  MoveL 6472 to (3.7, 324.47, -39.12) mm, rotated rx -180 ry 0 rz 0.01 deg; joints [44.471, -46.671, 108.236, -132.07, 70.721, 160.68]
  MoveL 6473 to (-1.54, 328.5, -39.37) mm, rotated rx 180 ry 0 rz 0.01 deg; joints [44.44, -46.388, 107.644, -132.02, 70.503, 160.447]
  MoveL 6474 to (0.05, 334.91, -39.61) mm, rotated rx -180 ry 0 rz 0.01 deg; joints [44.663, -46.238, 107.338, -131.758, 70.479, 160.247]
  MoveL 6475 to (6.56, 336.02, -39.86) mm, rotated rx 180 ry 0 rz 0.01 deg; joints [44.874, -46.386, 107.685, -131.602, 70.686, 160.333]
  MoveL 6476 to (10.19, 330.5, -40.1) mm, rotated rx -180 ry 0 rz 0.01 deg; joints [44.821, -46.638, 108.266, -131.74, 70.887, 160.611]
  MoveL 6477 to (6.58, 324.97, -40.35) mm, rotated rx -180 ry 0 rz 0.01 deg; joints [44.566, -46.676, 108.384, -132.014, 70.85, 160.76]
  MoveL 6478 to (0.07, 326.05, -40.59) mm, rotated rx 180 ry 0 rz 0.01 deg; joints [44.416, -46.439, 107.896, -132.097, 70.629, 160.613]
  MoveL 6479 to (-1.55, 332.45, -40.83) mm, rotated rx -180 ry 0 rz 0.01 deg; joints [44.551, -46.195, 107.385, -131.893, 70.498, 160.357]
  MoveL 6480 to (3.67, 336.5, -41.08) mm, rotated rx 180 ry 0 rz 0.01 deg; joints [44.808, -46.221, 107.462, -131.652, 70.625, 160.31]
  MoveL 6481 to (9.47, 333.34, -41.32) mm, rotated rx 180 ry 0 rz 0.01 deg; joints [44.881, -46.469, 108.034, -131.664, 70.865, 160.541]
  MoveL 6482 to (8.9, 326.76, -41.57) mm, rotated rx -180 ry 0 rz 0.01 deg; joints [44.681, -46.627, 108.413, -131.919, 70.943, 160.783]
  MoveL 6483 to (2.64, 324.65, -41.81) mm, rotated rx -180 ry 0 rz 0.01 deg; joints [44.448, -46.489, 108.144, -132.116, 70.773, 160.758]
  MoveL 6484 to (-1.8, 329.53, -42.05) mm, rotated rx -180 ry 0 rz 0.01 deg; joints [44.463, -46.205, 107.548, -132.02, 70.569, 160.507]
  MoveL 6485 to (0.89, 335.56, -42.3) mm, rotated rx -180 ry 0 rz 0.01 deg; joints [44.706, -46.1, 107.337, -131.752, 70.586, 160.342]
  MoveL 6486 to (7.49, 335.51, -42.54) mm, rotated rx -180 ry 0 rz 0.01 deg; joints [44.887, -46.283, 107.763, -131.636, 70.812, 160.472]
  MoveL 6487 to (10.09, 329.44, -42.79) mm, rotated rx 180 ry 0 rz 0.01 deg; joints [44.79, -46.519, 108.314, -131.814, 70.986, 160.753]
  MoveL 6488 to (5.57, 324.62, -43.03) mm, rotated rx -180 ry 0 rz 0.01 deg; joints [44.529, -46.51, 108.327, -132.078, 70.91, 160.858]
  MoveL 6489 to (-0.65, 326.84, -43.27) mm, rotated rx 180 ry 0 rz 0.01 deg; joints [44.419, -46.25, 107.786, -132.114, 70.683, 160.674]
  MoveL 6490 to (-1.12, 333.42, -43.52) mm, rotated rx 180 ry 0 rz 0.01 deg; joints [44.591, -46.035, 107.338, -131.883, 70.588, 160.432]
  MoveL 6491 to (4.73, 336.49, -43.76) mm, rotated rx -180 ry 0 rz 0.01 deg; joints [44.838, -46.108, 107.517, -131.666, 70.748, 160.433]
  MoveL 6492 to (9.89, 332.36, -44.01) mm, rotated rx -180 ry 0 rz 0.01 deg; joints [44.866, -46.364, 108.109, -131.725, 70.98, 160.688]
  MoveL 6493 to (8.17, 325.99, -44.25) mm, rotated rx 180 ry 0 rz 0.01 deg; joints [44.64, -46.481, 108.401, -131.995, 71.018, 160.902]
  MoveL 6494 to (1.64, 325, -44.49) mm, rotated rx -180 ry 0 rz 0.01 deg; joints [44.431, -46.303, 108.043, -132.155, 70.824, 160.83]
  MoveL 6495 to (-1.88, 330.59, -44.74) mm, rotated rx -180 ry 0 rz 0.01 deg; joints [44.492, -46.027, 107.461, -132.016, 70.64, 160.569]
  MoveL 6496 to (1.83, 336.06, -44.98) mm, rotated rx 180 ry 0 rz 0.01 deg; joints [44.747, -45.968, 107.352, -131.75, 70.698, 160.444]
  MoveL 6497 to (8.33, 334.84, -45.23) mm, rotated rx 180 ry 0 rz 0.01 deg; joints [44.893, -46.181, 107.845, -131.678, 70.936, 160.616]
  MoveL 6498 to (9.82, 328.41, -45.47) mm, rotated rx 180 ry 0 rz 0.01 deg; joints [44.754, -46.394, 108.347, -131.89, 71.08, 160.89]
  MoveL 6499 to (4.52, 324.47, -45.71) mm, rotated rx -180 ry 0 rz 0.01 deg; joints [44.496, -46.337, 108.255, -132.136, 70.967, 160.949]
  MoveL 6500 to (-1.22, 327.74, -45.96) mm, rotated rx -180 ry 0 rz 0.01 deg; joints [44.43, -46.062, 107.678, -132.124, 70.741, 160.734]
  MoveL 6501 to (-0.52, 334.31, -46.2) mm, rotated rx 180 ry 0 rz 0.01 deg; joints [44.633, -45.883, 107.306, -131.872, 70.683, 160.513]
  MoveL 6502 to (5.78, 336.3, -46.45) mm, rotated rx -180 ry 0 rz 0.01 deg; joints [44.863, -45.998, 107.582, -131.687, 70.872, 160.563]
  MoveL 6503 to (10.13, 331.32, -46.69) mm, rotated rx 180 ry 0 rz 0.01 deg; joints [44.845, -46.254, 108.175, -131.792, 71.09, 160.835]
  MoveL 6504 to (7.31, 325.35, -46.93) mm, rotated rx 180 ry 0 rz 0.01 deg; joints [44.599, -46.327, 108.372, -132.067, 71.087, 161.013]
  MoveL 6505 to (0.71, 325.53, -47.18) mm, rotated rx 180 ry 0 rz 0.01 deg; joints [44.422, -46.115, 107.935, -132.185, 70.875, 160.897]
  MoveL 6506 to (-1.76, 331.65, -47.42) mm, rotated rx 180 ry 0 rz 0.01 deg; joints [44.525, -45.855, 107.387, -132.008, 70.717, 160.635]
  MoveL 6507 to (2.85, 336.38, -47.67) mm, rotated rx -180 ry 0 rz 0.01 deg; joints [44.785, -45.844, 107.382, -131.753, 70.814, 160.553]
  MoveL 6508 to (9.03, 334.04, -47.91) mm, rotated rx -180 ry 0 rz 0.01 deg; joints [44.891, -46.078, 107.926, -131.728, 71.057, 160.761]
  MoveL 6509 to (9.36, 327.44, -48.15) mm, rotated rx -180 ry 0 rz 0.01 deg; joints [44.715, -46.261, 108.364, -131.966, 71.166, 161.02]
  MoveL 6510 to (3.45, 324.5, -48.4) mm, rotated rx 180 ry 0 rz 0.01 deg; joints [44.469, -46.158, 108.17, -132.188, 71.02, 161.031]
  MoveL 6511 to (-1.62, 328.73, -48.64) mm, rotated rx -180 ry 0 rz 0.01 deg; joints [44.448, -45.876, 107.575, -132.128, 70.802, 160.792]
  MoveL 6512 to (0.23, 335.07, -48.89) mm, rotated rx 180 ry 0 rz 0.01 deg; joints [44.676, -45.738, 107.29, -131.864, 70.785, 160.6]
  MoveL 6513 to (6.78, 335.92, -49.13) mm, rotated rx 180 ry 0 rz 0.01 deg; joints [44.881, -45.893, 107.655, -131.715, 70.997, 160.698]
  MoveL 6514 to (10.18, 330.26, -49.38) mm, rotated rx 180 ry 0 rz 0.01 deg; joints [44.818, -46.139, 108.231, -131.862, 71.195, 160.978]
  MoveL 6515 to (6.36, 324.87, -49.62) mm, rotated rx -180 ry 0 rz 0.01 deg; joints [44.56, -46.165, 108.325, -132.134, 71.151, 161.117]
  MoveL 6516 to (-0.11, 326.22, -49.86) mm, rotated rx 180 ry 0 rz 0.01 deg; joints [44.419, -45.925, 107.824, -132.208, 70.926, 160.959]
  MoveL 6517 to (-1.47, 332.68, -50.11) mm, rotated rx -180 ry 0 rz 0.01 deg; joints [44.563, -45.689, 107.325, -131.997, 70.801, 160.704]
  MoveL 6518 to (3.91, 336.51, -50.35) mm, rotated rx -180 ry 0 rz 0.01 deg; joints [44.819, -45.725, 107.426, -131.761, 70.934, 160.67]
  MoveL 6519 to (9.58, 333.13, -50.6) mm, rotated rx 180 ry 0 rz 0.01 deg; joints [44.882, -45.974, 108.003, -131.783, 71.175, 160.908]
  MoveL 6520 to (8.75, 326.57, -50.84) mm, rotated rx 180 ry 0 rz 0.01 deg; joints [44.675, -46.12, 108.363, -132.042, 71.246, 161.144]
  MoveL 6521 to (2.41, 324.71, -51.08) mm, rotated rx 180 ry 0 rz 0.01 deg; joints [44.447, -45.974, 108.073, -132.231, 71.071, 161.106]
  MoveL 6522 to (-1.84, 329.77, -51.33) mm, rotated rx 180 ry 0 rz 0.01 deg; joints [44.472, -45.694, 107.479, -132.126, 70.868, 160.852]
  MoveL 6523 to (1.1, 335.69, -51.57) mm, rotated rx 180 ry 0 rz 0.01 deg; joints [44.718, -45.6, 107.291, -131.858, 70.892, 160.695]
  MoveL 6524 to (7.69, 335.37, -51.82) mm, rotated rx 180 ry 0 rz 0.01 deg; joints [44.892, -45.789, 107.733, -131.751, 71.122, 160.837]
  MoveL 6525 to (10.05, 329.2, -52.06) mm, rotated rx 180 ry 0 rz 0.01 deg; joints [44.785, -46.018, 108.273, -131.936, 71.293, 161.118]
  MoveL 6526 to (5.34, 324.57, -52.3) mm, rotated rx 180 ry 0 rz 0.01 deg; joints [44.524, -45.997, 108.263, -132.197, 71.209, 161.211]
  MoveL 6527 to (-0.79, 327.03, -52.55) mm, rotated rx -180 ry 0 rz 0.01 deg; joints [44.425, -45.735, 107.712, -132.222, 70.98, 161.018]
  MoveL 6528 to (-0.99, 333.63, -52.79) mm, rotated rx -180 ry 0 rz 0.01 deg; joints [44.604, -45.53, 107.279, -131.986, 70.891, 160.779]
  MoveL 6529 to (4.97, 336.46, -53.04) mm, rotated rx -180 ry 0 rz 0.01 deg; joints [44.848, -45.612, 107.482, -131.776, 71.057, 160.793]
  MoveL 6530 to (9.96, 332.13, -53.28) mm, rotated rx 180 ry 0 rz 0.01 deg; joints [44.865, -45.866, 108.075, -131.845, 71.289, 161.054]
  MoveL 6531 to (7.98, 325.83, -53.52) mm, rotated rx 180 ry 0 rz 0.01 deg; joints [44.634, -45.972, 108.346, -132.116, 71.32, 161.26]
  MoveL 6532 to (1.42, 325.11, -53.77) mm, rotated rx 180 ry 0 rz 0.01 deg; joints [44.432, -45.787, 107.968, -132.267, 71.12, 161.176]
  MoveL 6533 to (-1.87, 330.84, -54.01) mm, rotated rx 180 ry 0 rz 0.01 deg; joints [44.502, -45.517, 107.393, -132.12, 70.94, 160.913]
  MoveL 6534 to (2.06, 336.15, -54.26) mm, rotated rx -180 ry 0 rz 0.01 deg; joints [44.759, -45.469, 107.307, -131.856, 71.005, 160.798]
  MoveL 6535 to (8.5, 334.67, -54.5) mm, rotated rx 180 ry 0 rz 0.01 deg; joints [44.896, -45.685, 107.812, -131.794, 71.246, 160.98]
  MoveL 6536 to (8.17, 335.16, -54.5) mm, rotated rx -180 ry 0 rz 0.01 deg; joints [44.9, -45.662, 107.76, -131.782, 71.228, 160.956]
  MoveL 6537 to (9.9, 336.02, -54.5) mm, rotated rx 180 ry 0 rz 0.01 deg; joints [44.973, -45.688, 107.816, -131.718, 71.273, 160.956]
  MoveL 6538 to (10.07, 335.56, -54.5) mm, rotated rx -180 ry 0 rz 0.01 deg; joints [44.965, -45.706, 107.857, -131.732, 71.285, 160.976]
  MoveL 6539 to (10.27, 334.35, -54.5) mm, rotated rx -180 ry 0 rz 0.01 deg; joints [44.936, -45.745, 107.946, -131.772, 71.308, 161.025]
  MoveL 6540 to (10.27, 32.01, -54.5) mm, rotated rx 180 ry 0 rz 0.01 deg; joints [35.147, -52.794, 124.522, -143.55, 75.758, 170.644]
  MoveL 6541 to (9.41, 35.75, -54.5) mm, rotated rx -180 ry 0 rz 0.01 deg; joints [35.264, -52.7, 124.291, -143.411, 75.67, 170.53]
  MoveL 6542 to (9.3, 36.12, -54.5) mm, rotated rx 180 ry 0 rz 0.01 deg; joints [35.275, -52.689, 124.267, -143.398, 75.66, 170.518]
  MoveL 6543 to (8.81, 37.5, -54.5) mm, rotated rx -180 ry 0 rz 0.01 deg; joints [35.313, -52.65, 124.17, -143.351, 75.621, 170.473]
  MoveL 6544 to (8.66, 37.84, -54.5) mm, rotated rx 180 ry 0 rz 0.01 deg; joints [35.321, -52.639, 124.145, -143.34, 75.611, 170.462]
  MoveL 6545 to (8, 39.21, -54.5) mm, rotated rx -180 ry 0 rz 0.01 deg; joints [35.355, -52.595, 124.036, -143.296, 75.566, 170.414]
  MoveL 6546 to (7.87, 39.46, -54.5) mm, rotated rx -180 ry 0 rz 0.01 deg; joints [35.36, -52.586, 124.017, -143.289, 75.558, 170.405]
  MoveL 6547 to (2.64, 48.31, -54.5) mm, rotated rx -180 ry 0 rz 0.01 deg; joints [35.549, -52.271, 123.255, -143.028, 75.238, 170.078]
  MoveL 6548 to (2.37, 48.71, -54.5) mm, rotated rx 180 ry 0 rz 0.01 deg; joints [35.556, -52.255, 123.218, -143.017, 75.222, 170.063]
  MoveL 6549 to (1.13, 50.25, -54.5) mm, rotated rx -180 ry 0 rz 0.01 deg; joints [35.58, -52.191, 123.063, -142.978, 75.154, 170]
  MoveL 6550 to (0.8, 50.61, -54.5) mm, rotated rx 180 ry 0 rz 0.01 deg; joints [35.585, -52.175, 123.025, -142.97, 75.137, 169.985]
  MoveL 6551 to (0, 51.35, -54.5) mm, rotated rx 180 ry 0 rz 0.01 deg; joints [35.591, -52.138, 122.937, -142.955, 75.098, 169.952]
  MoveL 6552 to (-1.84, 53.24, -54.5) mm, rotated rx 180 ry 0 rz 0.01 deg; joints [35.612, -52.049, 122.725, -142.915, 75.004, 169.869]
  MoveL 6553 to (-1.94, 53.34, -54.5) mm, rotated rx -180 ry 0 rz 0.01 deg; joints [35.613, -52.044, 122.713, -142.912, 74.999, 169.865]
  MoveL 6554 to (-4.34, 55.6, -54.5) mm, rotated rx 180 ry 0 rz 0.01 deg; joints [35.632, -51.932, 122.447, -142.868, 74.88, 169.763]
  MoveL 6555 to (-4.53, 55.76, -54.5) mm, rotated rx -180 ry 0 rz 0.01 deg; joints [35.633, -51.924, 122.427, -142.865, 74.87, 169.755]
  MoveL 6556 to (-7.2, 57.93, -54.5) mm, rotated rx -180 ry 0 rz 0.01 deg; joints [35.643, -51.805, 122.146, -142.829, 74.743, 169.651]
  MoveL 6557 to (-7.35, 58.05, -54.5) mm, rotated rx 180 ry 0 rz 0.01 deg; joints [35.643, -51.799, 122.13, -142.827, 74.735, 169.645]
  MoveL 6558 to (-117.5, 137.2, -54.5) mm, rotated rx 180 ry 0 rz 0.01 deg; joints [35.648, -46.798, 110.617, -141.535, 69.59, 165.45]
  MoveL 6559 to (-117.96, 137.48, -54.5) mm, rotated rx -180 ry 0 rz 0.01 deg; joints [35.647, -46.777, 110.57, -141.531, 69.569, 165.433]
  MoveL 6560 to (-119.42, 138.21, -54.5) mm, rotated rx 180 ry 0 rz 0.01 deg; joints [35.636, -46.714, 110.427, -141.523, 69.504, 165.385]
  MoveL 6561 to (-120.06, 138.45, -54.5) mm, rotated rx -180 ry 0 rz 0.01 deg; joints [35.629, -46.688, 110.369, -141.523, 69.477, 165.366]
  MoveL 6562 to (-121.51, 138.84, -54.5) mm, rotated rx -180 ry 0 rz 0.01 deg; joints [35.608, -46.632, 110.245, -141.528, 69.417, 165.328]
  MoveL 6563 to (-122.11, 138.94, -54.5) mm, rotated rx -180 ry 0 rz 0.01 deg; joints [35.597, -46.61, 110.196, -141.533, 69.393, 165.314]
  MoveL 6564 to (-123.56, 139.06, -54.5) mm, rotated rx -180 ry 0 rz 0.01 deg; joints [35.567, -46.56, 110.085, -141.549, 69.337, 165.285]
  MoveL 6565 to (-124.2, 139.05, -54.5) mm, rotated rx -180 ry 0 rz 0.01 deg; joints [35.552, -46.54, 110.039, -141.559, 69.313, 165.274]
  MoveL 6566 to (-126.74, 138.78, -54.5) mm, rotated rx 180 ry 0 rz 0.01 deg; joints [35.484, -46.463, 109.87, -141.607, 69.222, 165.238]
  MoveL 6567 to (-127.23, 138.69, -54.5) mm, rotated rx -180 ry 0 rz 0.01 deg; joints [35.47, -46.449, 109.839, -141.618, 69.205, 165.232]
  MoveL 6568 to (-129.41, 138.12, -54.5) mm, rotated rx -180 ry 0 rz 0.01 deg; joints [35.401, -46.391, 109.711, -141.672, 69.131, 165.211]
  MoveL 6569 to (-129.67, 138.04, -54.5) mm, rotated rx 180 ry 0 rz 0.01 deg; joints [35.392, -46.384, 109.696, -141.679, 69.122, 165.209]
  MoveL 6570 to (-131.12, 137.53, -54.5) mm, rotated rx 180 ry 0 rz 0.01 deg; joints [35.342, -46.348, 109.617, -141.72, 69.074, 165.199]
  MoveL 6571 to (-131.37, 137.43, -54.5) mm, rotated rx 180 ry 0 rz 0.01 deg; joints [35.333, -46.342, 109.603, -141.728, 69.066, 165.198]
  MoveL 6572 to (-134.37, 136.1, -54.5) mm, rotated rx 180 ry 0 rz 0.01 deg; joints [35.221, -46.273, 109.453, -141.825, 68.971, 165.187]
  MoveL 6573 to (-134.69, 135.94, -54.5) mm, rotated rx -180 ry 0 rz 0.01 deg; joints [35.208, -46.266, 109.439, -141.836, 68.961, 165.187]
  MoveL 6574 to (-171.12, 114.98, -54.5) mm, rotated rx 180 ry 0 rz 0.01 deg; joints [33.707, -45.509, 107.806, -143.175, 67.848, 165.2]
  MoveL 6575 to (-171.78, 114.49, -54.5) mm, rotated rx 180 ry 0 rz 0.01 deg; joints [33.676, -45.497, 107.781, -143.204, 67.829, 165.204]
  MoveL 6576 to (-172.53, 113.77, -54.5) mm, rotated rx -180 ry 0 rz 0.01 deg; joints [33.636, -45.487, 107.761, -143.243, 67.809, 165.213]
  MoveC 6577 to (-172.87, 113.39, -54.5) mm, rotated rx -180 ry 0 rz 0.01 deg; joints [33.617, -45.484, 107.754, -143.262, 67.801, 165.219] to (-173.15, 112.97, -54.5) mm, rotated rx 180 ry 0 rz 0.01 deg; joints [33.597, -45.483, 107.754, -143.283, 67.796, 165.227]
  MoveL 6578 to (-173.64, 112.08, -54.5) mm, rotated rx 180 ry 0 rz 0.01 deg; joints [33.557, -45.486, 107.761, -143.325, 67.789, 165.246]
  MoveC 6579 to (-173.86, 111.61, -54.5) mm, rotated rx 180 ry 0 rz 0.01 deg; joints [33.537, -45.489, 107.768, -143.347, 67.787, 165.257] to (-174, 111.11, -54.5) mm, rotated rx -180 ry 0 rz 0.01 deg; joints [33.517, -45.495, 107.782, -143.37, 67.788, 165.27]
  MoveL 6580 to (-174.22, 110.02, -54.5) mm, rotated rx 180 ry 0 rz 0.01 deg; joints [33.477, -45.511, 107.82, -143.417, 67.794, 165.301]
  MoveC 6581 to (-174.29, 109.49, -54.5) mm, rotated rx 180 ry 0 rz 0.01 deg; joints [33.458, -45.52, 107.841, -143.44, 67.798, 165.316] to (-174.27, 108.95, -54.5) mm, rotated rx -180 ry 0 rz 0.01 deg; joints [33.44, -45.532, 107.87, -143.461, 67.806, 165.333]
  MoveL 6582 to (-174.14, 107.86, -54.5) mm, rotated rx -180 ry 0 rz 0.01 deg; joints [33.408, -45.56, 107.933, -143.504, 67.826, 165.37]
  MoveC 6583 to (-174.03, 107.32, -54.5) mm, rotated rx -180 ry 0 rz 0.01 deg; joints [33.392, -45.576, 107.969, -143.525, 67.837, 165.389] to (-173.83, 106.8, -54.5) mm, rotated rx -180 ry 0 rz 0.01 deg; joints [33.379, -45.594, 108.009, -143.544, 67.852, 165.408]
  MoveL 6584 to (-173.32, 105.74, -54.5) mm, rotated rx -180 ry 0 rz 0.01 deg; joints [33.355, -45.634, 108.1, -143.581, 67.886, 165.45]
  MoveC 6585 to (-173.06, 105.29, -54.5) mm, rotated rx -180 ry 0 rz 0.01 deg; joints [33.346, -45.652, 108.142, -143.596, 67.903, 165.469] to (-172.73, 104.88, -54.5) mm, rotated rx 180 ry 0 rz 0.01 deg; joints [33.34, -45.673, 108.187, -143.609, 67.921, 165.488]
  MoveL 6586 to (-172.05, 104.16, -54.5) mm, rotated rx 180 ry 0 rz 0.01 deg; joints [33.331, -45.711, 108.273, -143.629, 67.957, 165.522]
  MoveL 6587 to (-171.28, 103.56, -54.5) mm, rotated rx -180 ry 0 rz 0.01 deg; joints [33.328, -45.75, 108.36, -143.644, 67.995, 165.554]
  MoveL 6588 to (-55.84, 36.98, -54.5) mm, rotated rx 180 ry 0 rz 0.01 deg; joints [33.667, -50.782, 119.826, -144.62, 73.292, 169.428]
  MoveL 6589 to (-63.76, 23.29, -54.5) mm, rotated rx 180 ry 0 rz 0.01 deg; joints [32.98, -50.8, 119.9, -145.332, 73.197, 169.672]
  MoveL 6590 to (-178.74, 89.79, -54.5) mm, rotated rx -180 ry 0 rz 0.01 deg; joints [32.71, -45.788, 108.472, -144.303, 67.887, 165.848]
  MoveL 6591 to (-179.27, 90.04, -54.5) mm, rotated rx 180 ry 0 rz 0.01 deg; joints [32.707, -45.765, 108.42, -144.299, 67.863, 165.831]
  MoveL 6592 to (-180.24, 90.4, -54.5) mm, rotated rx -180 ry 0 rz 0.01 deg; joints [32.698, -45.724, 108.329, -144.297, 67.82, 165.803]
  MoveC 6593 to (-180.73, 90.53, -54.5) mm, rotated rx 180 ry 0 rz 0.01 deg; joints [32.693, -45.704, 108.285, -144.297, 67.799, 165.79] to (-181.24, 90.6, -54.5) mm, rotated rx 180 ry 0 rz 0.01 deg; joints [32.684, -45.685, 108.244, -144.301, 67.778, 165.779]
  MoveL 6594 to (-182.28, 90.65, -54.5) mm, rotated rx -180 ry 0 rz 0.01 deg; joints [32.664, -45.649, 108.162, -144.311, 67.737, 165.759]
  MoveC 6595 to (-182.79, 90.64, -54.5) mm, rotated rx 180 ry 0 rz 0.01 deg; joints [32.652, -45.631, 108.124, -144.318, 67.716, 165.751] to (-183.29, 90.55, -54.5) mm, rotated rx -180 ry 0 rz 0.01 deg; joints [32.638, -45.616, 108.09, -144.328, 67.698, 165.745]
  MoveL 6596 to (-184.32, 90.28, -54.5) mm, rotated rx -180 ry 0 rz 0.01 deg; joints [32.608, -45.586, 108.025, -144.351, 67.661, 165.735]
  MoveC 6597 to (-184.81, 90.11, -54.5) mm, rotated rx 180 ry 0 rz 0.01 deg; joints [32.592, -45.573, 107.996, -144.364, 67.644, 165.732] to (-185.27, 89.87, -54.5) mm, rotated rx -180 ry 0 rz 0.01 deg; joints [32.574, -45.562, 107.973, -144.38, 67.629, 165.731]
  MoveL 6598 to (-186.19, 89.29, -54.5) mm, rotated rx 180 ry 0 rz 0.01 deg; joints [32.535, -45.543, 107.931, -144.415, 67.6, 165.733]
  MoveL 6599 to (-186.72, 88.88, -54.5) mm, rotated rx 180 ry 0 rz 0.01 deg; joints [32.51, -45.533, 107.911, -144.438, 67.585, 165.736]
  MoveL 6600 to (-186.93, 88.67, -54.5) mm, rotated rx 180 ry 0 rz 0.01 deg; joints [32.499, -45.53, 107.904, -144.449, 67.579, 165.739]
  MoveL 6601 to (-187.39, 88.14, -54.5) mm, rotated rx 180 ry 0 rz 0.01 deg; joints [32.471, -45.526, 107.896, -144.477, 67.568, 165.747]
  MoveL 6602 to (-188.03, 87.2, -54.5) mm, rotated rx 180 ry 0 rz 0.01 deg; joints [32.427, -45.523, 107.892, -144.523, 67.555, 165.765]
  MoveC 6603 to (-188.3, 86.74, -54.5) mm, rotated rx 180 ry 0 rz 0.01 deg; joints [32.406, -45.524, 107.894, -144.545, 67.551, 165.774] to (-188.48, 86.25, -54.5) mm, rotated rx -180 ry 0 rz 0.01 deg; joints [32.386, -45.527, 107.903, -144.568, 67.55, 165.786]
  MoveL 6604 to (-188.77, 85.29, -54.5) mm, rotated rx -180 ry 0 rz 0.01 deg; joints [32.347, -45.538, 107.928, -144.611, 67.551, 165.811]
  MoveL 6605 to (-188.91, 84.32, -54.5) mm, rotated rx 180 ry 0 rz 0.01 deg; joints [32.312, -45.553, 107.964, -144.653, 67.558, 165.838]
  MoveL 6606 to (-188.88, 42.24, -54.5) mm, rotated rx 180 ry 0 rz 0.01 deg; joints [30.889, -46.405, 109.934, -146.395, 68.114, 167.097]
  MoveL 6607 to (-188.87, 41.91, -54.5) mm, rotated rx -180 ry 0 rz 0.01 deg; joints [30.878, -46.412, 109.95, -146.409, 68.119, 167.107]
  MoveL 6608 to (-188.58, 39.01, -54.5) mm, rotated rx 180 ry 0 rz 0.01 deg; joints [30.784, -46.478, 110.104, -146.526, 68.169, 167.196]
  MoveL 6609 to (-188.54, 38.69, -54.5) mm, rotated rx 180 ry 0 rz 0.01 deg; joints [30.774, -46.486, 110.122, -146.539, 68.175, 167.206]
  MoveL 6610 to (-187.97, 35.79, -54.5) mm, rotated rx 180 ry 0 rz 0.01 deg; joints [30.686, -46.562, 110.296, -146.653, 68.235, 167.3]
  MoveL 6611 to (-187.88, 35.43, -54.5) mm, rotated rx 180 ry 0 rz 0.01 deg; joints [30.675, -46.572, 110.319, -146.666, 68.244, 167.312]
  MoveL 6612 to (-187.43, 33.98, -54.5) mm, rotated rx 180 ry 0 rz 0.01 deg; joints [30.635, -46.615, 110.419, -146.721, 68.281, 167.361]
  MoveL 6613 to (-187.31, 33.65, -54.5) mm, rotated rx -180 ry 0 rz 0.01 deg; joints [30.626, -46.626, 110.443, -146.734, 68.29, 167.373]
  MoveL 6614 to (-186.62, 32.06, -54.5) mm, rotated rx 180 ry 0 rz 0.01 deg; joints [30.585, -46.68, 110.566, -146.792, 68.338, 167.43]
  MoveL 6615 to (-186.43, 31.68, -54.5) mm, rotated rx 180 ry 0 rz 0.01 deg; joints [30.576, -46.693, 110.597, -146.805, 68.351, 167.444]
  MoveL 6616 to (-185.67, 30.38, -54.5) mm, rotated rx -180 ry 0 rz 0.01 deg; joints [30.546, -46.745, 110.714, -146.85, 68.398, 167.494]
  MoveL 6617 to (-185.34, 29.91, -54.5) mm, rotated rx 180 ry 0 rz 0.01 deg; joints [30.536, -46.765, 110.761, -146.866, 68.418, 167.513]
  MoveL 6618 to (-184.36, 28.74, -54.5) mm, rotated rx 180 ry 0 rz 0.01 deg; joints [30.516, -46.821, 110.887, -146.902, 68.472, 167.563]
  MoveL 6619 to (-183.78, 28.2, -54.5) mm, rotated rx 180 ry 0 rz 0.01 deg; joints [30.509, -46.851, 110.955, -146.918, 68.503, 167.588]
  MoveL 6620 to (-182.33, 27.14, -54.5) mm, rotated rx 180 ry 0 rz 0.01 deg; joints [30.502, -46.92, 111.112, -146.944, 68.574, 167.642]
  MoveL 6621 to (-181.72, 26.78, -54.5) mm, rotated rx 180 ry 0 rz 0.01 deg; joints [30.502, -46.948, 111.175, -146.952, 68.603, 167.663]
  MoveL 6622 to (-60.29, -28.09, -54.5) mm, rotated rx 180 ry 0 rz 0.01 deg; joints [31.142, -51.818, 122.383, -147.451, 74.067, 171.067]
  MoveL 6623 to (-60.24, -28.11, -54.5) mm, rotated rx 180 ry 0 rz 0.01 deg; joints [31.142, -51.82, 122.388, -147.451, 74.069, 171.068]
  MoveL 6624 to (-55.89, -30, -54.5) mm, rotated rx 180 ry 0 rz 0.01 deg; joints [31.171, -51.982, 122.771, -147.455, 74.26, 171.184]
  MoveL 6625 to (-55.59, -30.11, -54.5) mm, rotated rx 180 ry 0 rz 0.01 deg; joints [31.174, -51.993, 122.797, -147.455, 74.273, 171.191]
  MoveL 6626 to (-52.03, -31.27, -54.5) mm, rotated rx -180 ry 0 rz 0.01 deg; joints [31.212, -52.118, 123.094, -147.442, 74.424, 171.276]
  MoveL 6627 to (-341.51, -31.27, -54.5) mm, rotated rx -180 ry 0 rz 0.01 deg; joints [25.59, -42.149, 100.744, -150.865, 62.571, 166.683]
  MoveL 6628 to (-339.42, -30.62, -54.5) mm, rotated rx 180 ry 0 rz 0.01 deg; joints [25.646, -42.22, 100.898, -150.825, 62.657, 166.699]
  MoveL 6629 to (-339.24, -30.56, -54.5) mm, rotated rx -180 ry 0 rz 0.01 deg; joints [25.651, -42.226, 100.911, -150.821, 62.664, 166.701]
  MoveL 6630 to (-336.33, -29.47, -54.5) mm, rotated rx -180 ry 0 rz 0.01 deg; joints [25.735, -42.321, 101.115, -150.758, 62.781, 166.718]
  MoveL 6631 to (-336.13, -29.39, -54.5) mm, rotated rx -180 ry 0 rz 0.01 deg; joints [25.741, -42.328, 101.13, -150.753, 62.79, 166.719]
  MoveL 6632 to (-212.26, 26.52, -54.5) mm, rotated rx 180 ry 0 rz 0.01 deg; joints [29.878, -45.898, 108.843, -147.324, 67.376, 167.164]
  MoveL 6633 to (-211.79, 26.78, -54.5) mm, rotated rx 180 ry 0 rz 0.01 deg; joints [29.896, -45.91, 108.868, -147.308, 67.392, 167.164]
  MoveL 6634 to (-210.12, 27.88, -54.5) mm, rotated rx 180 ry 0 rz 0.01 deg; joints [29.967, -45.947, 108.948, -147.243, 67.446, 167.16]
  MoveL 6635 to (-209.55, 28.36, -54.5) mm, rotated rx -180 ry 0 rz 0.01 deg; joints [29.995, -45.958, 108.972, -147.216, 67.463, 167.156]
  MoveL 6636 to (-208.78, 29.16, -54.5) mm, rotated rx 180 ry 0 rz 0.01 deg; joints [30.038, -45.969, 108.996, -147.174, 67.484, 167.145]
  MoveL 6637 to (-208.44, 29.57, -54.5) mm, rotated rx 180 ry 0 rz 0.01 deg; joints [30.058, -45.973, 109.003, -147.153, 67.492, 167.139]
  MoveL 6638 to (-207.43, 31.01, -54.5) mm, rotated rx 180 ry 0 rz 0.01 deg; joints [30.128, -45.981, 109.017, -147.082, 67.514, 167.114]
  MoveL 6639 to (-207.11, 31.59, -54.5) mm, rotated rx 180 ry 0 rz 0.01 deg; joints [30.154, -45.981, 109.016, -147.054, 67.52, 167.102]
  MoveL 6640 to (-206.22, 33.63, -54.5) mm, rotated rx 180 ry 0 rz 0.01 deg; joints [30.242, -45.973, 108.994, -146.958, 67.53, 167.058]
  MoveL 6641 to (-206.08, 33.98, -54.5) mm, rotated rx 180 ry 0 rz 0.01 deg; joints [30.257, -45.97, 108.988, -146.942, 67.531, 167.05]
  MoveL 6642 to (-205.63, 35.43, -54.5) mm, rotated rx 180 ry 0 rz 0.01 deg; joints [30.316, -45.958, 108.957, -146.876, 67.53, 167.015]
  MoveL 6643 to (-205.54, 35.79, -54.5) mm, rotated rx 180 ry 0 rz 0.01 deg; joints [30.33, -45.954, 108.948, -146.86, 67.529, 167.006]
  MoveL 6644 to (-204.98, 38.69, -54.5) mm, rotated rx -180 ry 0 rz 0.01 deg; joints [30.441, -45.917, 108.861, -146.733, 67.514, 166.93]
  MoveL 6645 to (-204.93, 39.01, -54.5) mm, rotated rx -180 ry 0 rz 0.01 deg; joints [30.452, -45.913, 108.85, -146.719, 67.512, 166.922]
  MoveL 6646 to (-204.64, 41.91, -54.5) mm, rotated rx -180 ry 0 rz 0.01 deg; joints [30.557, -45.866, 108.741, -146.595, 67.486, 166.841]
  MoveL 6647 to (-204.63, 42.24, -54.5) mm, rotated rx -180 ry 0 rz 0.01 deg; joints [30.569, -45.86, 108.727, -146.581, 67.482, 166.832]
  MoveL 6648 to (-204.6, 84.32, -54.5) mm, rotated rx 180 ry 0 rz 0.01 deg; joints [31.985, -45.007, 106.761, -144.836, 66.934, 165.563]
  MoveL 6649 to (-204.74, 85.29, -54.5) mm, rotated rx 180 ry 0 rz 0.01 deg; joints [32.014, -44.982, 106.704, -144.797, 66.915, 165.53]
  MoveL 6650 to (-205.03, 86.25, -54.5) mm, rotated rx 180 ry 0 rz 0.01 deg; joints [32.04, -44.951, 106.635, -144.76, 66.891, 165.495]
  MoveC 6651 to (-205.22, 86.74, -54.5) mm, rotated rx 180 ry 0 rz 0.01 deg; joints [32.052, -44.934, 106.597, -144.742, 66.877, 165.476] to (-205.48, 87.2, -54.5) mm, rotated rx -180 ry 0 rz 0.01 deg; joints [32.062, -44.916, 106.554, -144.726, 66.861, 165.458]
  MoveL 6652 to (-206.12, 88.14, -54.5) mm, rotated rx -180 ry 0 rz 0.01 deg; joints [32.079, -44.873, 106.459, -144.695, 66.822, 165.417]
  MoveC 6653 to (-206.47, 88.57, -54.5) mm, rotated rx -180 ry 0 rz 0.01 deg; joints [32.086, -44.852, 106.411, -144.681, 66.803, 165.398] to (-206.89, 88.94, -54.5) mm, rotated rx 180 ry 0 rz 0.01 deg; joints [32.09, -44.829, 106.362, -144.671, 66.781, 165.379]
  MoveL 6654 to (-207.79, 89.61, -54.5) mm, rotated rx 180 ry 0 rz 0.01 deg; joints [32.094, -44.783, 106.259, -144.653, 66.736, 165.342]
  MoveC 6655 to (-208.22, 89.88, -54.5) mm, rotated rx -180 ry 0 rz 0.01 deg; joints [32.094, -44.762, 106.213, -144.646, 66.715, 165.326] to (-208.69, 90.09, -54.5) mm, rotated rx 180 ry 0 rz 0.01 deg; joints [32.091, -44.742, 106.166, -144.643, 66.694, 165.311]
  MoveL 6656 to (-209.59, 90.41, -54.5) mm, rotated rx -180 ry 0 rz 0.01 deg; joints [32.083, -44.703, 106.081, -144.64, 66.654, 165.285]
  MoveL 6657 to (-210.55, 90.6, -54.5) mm, rotated rx 180 ry 0 rz 0.01 deg; joints [32.069, -44.665, 105.998, -144.643, 66.613, 165.262]
  MoveL 6658 to (-211.59, 90.65, -54.5) mm, rotated rx -180 ry 0 rz 0.01 deg; joints [32.049, -44.627, 105.915, -144.652, 66.57, 165.242]
  MoveL 6659 to (-212.57, 90.56, -54.5) mm, rotated rx 180 ry 0 rz 0.01 deg; joints [32.026, -44.594, 105.843, -144.667, 66.532, 165.227]
  MoveL 6660 to (-213.53, 90.32, -54.5) mm, rotated rx -180 ry 0 rz 0.01 deg; joints [31.998, -44.566, 105.78, -144.687, 66.496, 165.217]
  MoveL 6661 to (-214.41, 89.96, -54.5) mm, rotated rx 180 ry 0 rz 0.01 deg; joints [31.969, -44.542, 105.728, -144.711, 66.466, 165.213]
  MoveL 6662 to (-329.75, 23.29, -54.5) mm, rotated rx 180 ry 0 rz 0.01 deg; joints [27.603, -41.584, 99.413, -148.476, 62.445, 165.215]
  MoveL 6663 to (-337.67, 36.98, -54.5) mm, rotated rx 180 ry 0 rz 0.01 deg; joints [27.914, -40.994, 98.113, -147.941, 61.929, 164.631]
  MoveL 6664 to (-222.23, 103.56, -54.5) mm, rotated rx 180 ry 0 rz 0.01 deg; joints [32.253, -43.972, 104.453, -144.233, 65.973, 164.642]
  MoveL 6665 to (-221.46, 104.16, -54.5) mm, rotated rx -180 ry 0 rz 0.01 deg; joints [32.288, -43.986, 104.484, -144.2, 65.996, 164.637]
  MoveL 6666 to (-220.79, 104.88, -54.5) mm, rotated rx 180 ry 0 rz 0.01 deg; joints [32.325, -43.995, 104.501, -144.164, 66.014, 164.627]
  MoveC 6667 to (-220.45, 105.29, -54.5) mm, rotated rx 180 ry 0 rz 0.01 deg; joints [32.345, -43.998, 104.507, -144.143, 66.022, 164.62] to (-220.19, 105.74, -54.5) mm, rotated rx -180 ry 0 rz 0.01 deg; joints [32.365, -43.997, 104.505, -144.122, 66.026, 164.61]
  MoveL 6668 to (-219.68, 106.8, -54.5) mm, rotated rx -180 ry 0 rz 0.01 deg; joints [32.41, -43.992, 104.492, -144.073, 66.033, 164.585]
  MoveC 6669 to (-219.49, 107.32, -54.5) mm, rotated rx -180 ry 0 rz 0.01 deg; joints [32.431, -43.988, 104.482, -144.049, 66.034, 164.572] to (-219.37, 107.86, -54.5) mm, rotated rx -180 ry 0 rz 0.01 deg; joints [32.451, -43.98, 104.464, -144.026, 66.031, 164.557]
  MoveL 6670 to (-219.25, 108.95, -54.5) mm, rotated rx -180 ry 0 rz 0.01 deg; joints [32.489, -43.961, 104.42, -143.98, 66.022, 164.524]
  MoveC 6671 to (-219.22, 109.49, -54.5) mm, rotated rx 180 ry 0 rz 0.01 deg; joints [32.507, -43.95, 104.395, -143.957, 66.016, 164.508] to (-219.29, 110.02, -54.5) mm, rotated rx 180 ry 0 rz 0.01 deg; joints [32.523, -43.936, 104.363, -143.936, 66.007, 164.489]
  MoveL 6672 to (-219.51, 111.11, -54.5) mm, rotated rx -180 ry 0 rz 0.01 deg; joints [32.553, -43.904, 104.292, -143.893, 65.983, 164.45]
  MoveC 6673 to (-219.65, 111.61, -54.5) mm, rotated rx 180 ry 0 rz 0.01 deg; joints [32.567, -43.888, 104.256, -143.874, 65.971, 164.431] to (-219.87, 112.08, -54.5) mm, rotated rx 180 ry 0 rz 0.01 deg; joints [32.577, -43.87, 104.215, -143.857, 65.956, 164.412]
  MoveL 6674 to (-220.37, 112.97, -54.5) mm, rotated rx -180 ry 0 rz 0.01 deg; joints [32.596, -43.833, 104.132, -143.826, 65.925, 164.375]
  MoveC 6675 to (-220.64, 113.39, -54.5) mm, rotated rx 180 ry 0 rz 0.01 deg; joints [32.604, -43.813, 104.089, -143.811, 65.908, 164.356] to (-220.98, 113.77, -54.5) mm, rotated rx -180 ry 0 rz 0.01 deg; joints [32.609, -43.793, 104.044, -143.8, 65.889, 164.338]
  MoveL 6676 to (-221.74, 114.49, -54.5) mm, rotated rx -180 ry 0 rz 0.01 deg; joints [32.616, -43.75, 103.949, -143.778, 65.849, 164.301]
  MoveL 6677 to (-222.39, 114.98, -54.5) mm, rotated rx 180 ry 0 rz 0.01 deg; joints [32.619, -43.716, 103.873, -143.764, 65.817, 164.273]
  MoveL 6678 to (-258.15, 135.55, -54.5) mm, rotated rx 180 ry 0 rz 0.01 deg; joints [32.546, -41.94, 99.976, -143.251, 64.089, 162.913]
  MoveL 6679 to (-258.3, 135.64, -54.5) mm, rotated rx -180 ry 0 rz 0.01 deg; joints [32.546, -41.933, 99.959, -143.248, 64.081, 162.907]
  MoveL 6680 to (-260.33, 136.67, -54.5) mm, rotated rx -180 ry 0 rz 0.01 deg; joints [32.538, -41.833, 99.741, -143.223, 63.984, 162.832]
  MoveL 6681 to (-260.65, 136.81, -54.5) mm, rotated rx -180 ry 0 rz 0.01 deg; joints [32.536, -41.818, 99.708, -143.22, 63.969, 162.821]
  MoveL 6682 to (-263.74, 138, -54.5) mm, rotated rx 180 ry 0 rz 0.01 deg; joints [32.511, -41.673, 99.394, -143.195, 63.825, 162.72]
  MoveL 6683 to (-264.11, 138.12, -54.5) mm, rotated rx -180 ry 0 rz 0.01 deg; joints [32.508, -41.657, 99.358, -143.194, 63.809, 162.709]
  MoveL 6684 to (-266.28, 138.69, -54.5) mm, rotated rx 180 ry 0 rz 0.01 deg; joints [32.482, -41.561, 99.151, -143.188, 63.711, 162.646]
  MoveL 6685 to (-266.73, 138.77, -54.5) mm, rotated rx -180 ry 0 rz 0.01 deg; joints [32.476, -41.543, 99.11, -143.188, 63.691, 162.634]
  MoveL 6686 to (-268.9, 139.04, -54.5) mm, rotated rx 180 ry 0 rz 0.01 deg; joints [32.441, -41.454, 98.918, -143.194, 63.597, 162.582]
  MoveL 6687 to (-269.44, 139.06, -54.5) mm, rotated rx 180 ry 0 rz 0.01 deg; joints [32.431, -41.433, 98.873, -143.197, 63.575, 162.57]
  MoveL 6688 to (-270.89, 139, -54.5) mm, rotated rx -180 ry 0 rz 0.01 deg; joints [32.401, -41.379, 98.757, -143.211, 63.515, 162.543]
  MoveL 6689 to (-271.45, 138.94, -54.5) mm, rotated rx -180 ry 0 rz 0.01 deg; joints [32.387, -41.359, 98.714, -143.218, 63.493, 162.535]
  MoveL 6690 to (-272.9, 138.63, -54.5) mm, rotated rx -180 ry 0 rz 0.01 deg; joints [32.349, -41.311, 98.611, -143.242, 63.436, 162.516]
  MoveL 6691 to (-273.61, 138.41, -54.5) mm, rotated rx -180 ry 0 rz 0.01 deg; joints [32.328, -41.29, 98.565, -143.256, 63.409, 162.51]
  MoveL 6692 to (-275.06, 137.75, -54.5) mm, rotated rx 180 ry 0 rz 0.01 deg; joints [32.279, -41.25, 98.479, -143.295, 63.357, 162.503]
  MoveL 6693 to (-275.64, 137.42, -54.5) mm, rotated rx -180 ry 0 rz 0.01 deg; joints [32.257, -41.235, 98.449, -143.313, 63.337, 162.503]
  MoveL 6694 to (-382.15, 60.93, -54.5) mm, rotated rx -180 ry 0 rz 0.01 deg; joints [27.926, -38.662, 93.057, -147.11, 59.635, 162.949]
  MoveL 6695 to (-387.52, 56.99, -54.5) mm, rotated rx 180 ry 0 rz 0.01 deg; joints [27.713, -38.519, 92.757, -147.295, 59.436, 162.972]
  MoveL 6696 to (-387.77, 56.79, -54.5) mm, rotated rx 180 ry 0 rz 0.01 deg; joints [27.703, -38.512, 92.744, -147.304, 59.427, 162.973]
  MoveL 6697 to (-390.95, 53.96, -54.5) mm, rotated rx 180 ry 0 rz 0.01 deg; joints [27.561, -38.437, 92.588, -147.434, 59.315, 163.004]
  MoveL 6698 to (-391.17, 53.75, -54.5) mm, rotated rx 180 ry 0 rz 0.01 deg; joints [27.551, -38.432, 92.578, -147.444, 59.307, 163.007]
  MoveL 6699 to (-392.89, 51.93, -54.5) mm, rotated rx -180 ry 0 rz 0.01 deg; joints [27.465, -38.398, 92.508, -147.527, 59.25, 163.033]
  MoveL 6700 to (-394, 50.94, -54.5) mm, rotated rx -180 ry 0 rz 0.01 deg; joints [27.416, -38.371, 92.452, -147.572, 59.21, 163.044]
  MoveL 6701 to (-394.39, 50.54, -54.5) mm, rotated rx 180 ry 0 rz 0.01 deg; joints [27.397, -38.363, 92.436, -147.59, 59.197, 163.049]
  MoveL 6702 to (-395.86, 48.73, -54.5) mm, rotated rx -180 ry 0 rz 0.01 deg; joints [27.316, -38.338, 92.387, -147.672, 59.151, 163.081]
  MoveL 6703 to (-396.11, 48.38, -54.5) mm, rotated rx -180 ry 0 rz 0.01 deg; joints [27.301, -38.335, 92.38, -147.688, 59.143, 163.088]
  MoveL 6704 to (-397.02, 46.93, -54.5) mm, rotated rx 180 ry 0 rz 0.01 deg; joints [27.241, -38.327, 92.366, -147.752, 59.119, 163.118]
  MoveL 6705 to (-397.07, 46.84, -54.5) mm, rotated rx 180 ry 0 rz 0.01 deg; joints [27.237, -38.327, 92.365, -147.756, 59.118, 163.12]
  MoveL 6706 to (-401.78, 38.75, -54.5) mm, rotated rx 180 ry 0 rz 0.01 deg; joints [26.906, -38.295, 92.312, -148.117, 58.996, 163.299]
  MoveL 6707 to (-402, 38.3, -54.5) mm, rotated rx -180 ry 0 rz 0.01 deg; joints [26.888, -38.295, 92.312, -148.137, 58.991, 163.31]
  MoveL 6708 to (-402.68, 36.58, -54.5) mm, rotated rx -180 ry 0 rz 0.01 deg; joints [26.822, -38.302, 92.33, -148.213, 58.98, 163.355]
  MoveL 6709 to (-402.83, 36.1, -54.5) mm, rotated rx 180 ry 0 rz 0.01 deg; joints [26.805, -38.305, 92.338, -148.233, 58.979, 163.368]
  MoveL 6710 to (-403.78, 32.04, -54.5) mm, rotated rx 180 ry 0 rz 0.01 deg; joints [26.661, -38.349, 92.439, -148.411, 58.983, 163.487]
  MoveL 6711 to (-403.79, 333.8, -54.5) mm, rotated rx -180 ry 0 rz 0.01 deg; joints [35.419, -30.182, 74.721, -134.972, 55.031, 151.097]
  MoveL 6712 to (-403.73, 334.87, -54.5) mm, rotated rx 180 ry 0 rz 0.01 deg; joints [35.448, -30.148, 74.648, -134.922, 55.018, 151.045]
  MoveL 6713 to (-403.53, 335.74, -54.5) mm, rotated rx 180 ry 0 rz 0.01 deg; joints [35.474, -30.127, 74.604, -134.883, 55.015, 151.009]
  MoveL 6714 to (-403.42, 336, -54.5) mm, rotated rx -180 ry 0 rz 0.01 deg; joints [35.484, -30.124, 74.597, -134.871, 55.017, 150.999]
  MoveL 6715 to (-403.21, 336.31, -54.5) mm, rotated rx 180 ry 0 rz 0.01 deg; joints [35.496, -30.124, 74.596, -134.858, 55.022, 150.991]
  MoveL 6716 to (-400.95, 338.6, -54.5) mm, rotated rx -180 ry 0 rz 0.01 deg; joints [35.598, -30.156, 74.66, -134.766, 55.097, 150.956]
  MoveL 6717 to (-400.6, 338.83, -54.5) mm, rotated rx 180 ry 0 rz 0.01 deg; joints [35.611, -30.166, 74.68, -134.757, 55.11, 150.957]
  MoveL 6718 to (-400.13, 339.01, -54.5) mm, rotated rx 180 ry 0 rz 0.01 deg; joints [35.624, -30.182, 74.715, -134.752, 55.13, 150.965]
  MoveL 6719 to (-398.92, 339.2, -54.5) mm, rotated rx -180 ry 0 rz 0.01 deg; joints [35.652, -30.236, 74.826, -134.752, 55.185, 150.997]
  MoveL 6720 to (-213.44, 339.2, -54.5) mm, rotated rx -180 ry 0 rz 0.01 deg; joints [39.472, -38.205, 91.627, -134.561, 63.179, 156.254]
  MoveL 6721 to (-213.6, 339.17, -54.5) mm, rotated rx -180 ry 0 rz 0.01 deg; joints [39.467, -38.2, 91.617, -134.563, 63.174, 156.252]
  MoveL 6722 to (-214.68, 338.87, -54.5) mm, rotated rx 180 ry 0 rz 0.01 deg; joints [39.435, -38.168, 91.549, -134.583, 63.135, 156.238]
  MoveL 6723 to (-215.27, 338.65, -54.5) mm, rotated rx -180 ry 0 rz 0.01 deg; joints [39.416, -38.153, 91.516, -134.596, 63.114, 156.233]
  MoveL 6724 to (-225.79, 333.59, -54.5) mm, rotated rx -180 ry 0 rz 0.01 deg; joints [39.043, -37.906, 90.999, -134.876, 62.765, 156.193]
  MoveL 6725 to (-226.17, 333.38, -54.5) mm, rotated rx 180 ry 0 rz 0.01 deg; joints [39.029, -37.898, 90.982, -134.887, 62.753, 156.193]
  MoveL 6726 to (-227.62, 332.44, -54.5) mm, rotated rx 180 ry 0 rz 0.01 deg; joints [38.971, -37.871, 90.926, -134.936, 62.708, 156.197]
  MoveL 6727 to (-228.09, 332.08, -54.5) mm, rotated rx -180 ry 0 rz 0.01 deg; joints [38.951, -37.864, 90.912, -134.954, 62.694, 156.201]
  MoveL 6728 to (-236.32, 324.39, -54.5) mm, rotated rx 180 ry 0 rz 0.01 deg; joints [38.559, -37.779, 90.742, -135.322, 62.468, 156.322]
  MoveL 6729 to (-236.66, 324.02, -54.5) mm, rotated rx 180 ry 0 rz 0.01 deg; joints [38.542, -37.777, 90.739, -135.34, 62.459, 156.329]
  MoveL 6730 to (-238.09, 322.2, -54.5) mm, rotated rx -180 ry 0 rz 0.01 deg; joints [38.46, -37.776, 90.739, -135.423, 62.426, 156.37]
  MoveL 6731 to (-238.39, 321.77, -54.5) mm, rotated rx 180 ry 0 rz 0.01 deg; joints [38.442, -37.778, 90.743, -135.443, 62.42, 156.381]
  MoveL 6732 to (-243.72, 312.34, -54.5) mm, rotated rx -180 ry 0 rz 0.01 deg; joints [38.066, -37.853, 90.916, -135.864, 62.332, 156.641]
  MoveL 6733 to (-243.93, 311.9, -54.5) mm, rotated rx 180 ry 0 rz 0.01 deg; joints [38.049, -37.857, 90.927, -135.884, 62.33, 156.654]
  MoveL 6734 to (-244.63, 310.08, -54.5) mm, rotated rx -180 ry 0 rz 0.01 deg; joints [37.984, -37.884, 90.986, -135.963, 62.326, 156.711]
  MoveL 6735 to (-244.78, 309.58, -54.5) mm, rotated rx -180 ry 0 rz 0.01 deg; joints [37.967, -37.893, 91.006, -135.984, 62.326, 156.728]
  MoveL 6736 to (-245.07, 308.25, -54.5) mm, rotated rx -180 ry 0 rz 0.01 deg; joints [37.923, -37.921, 91.067, -136.041, 62.332, 156.776]
  MoveL 6737 to (-245.79, 305.84, -54.5) mm, rotated rx -180 ry 0 rz 0.01 deg; joints [37.841, -37.964, 91.163, -136.145, 62.336, 156.857]
  MoveL 6738 to (-245.85, 305.62, -54.5) mm, rotated rx -180 ry 0 rz 0.01 deg; joints [37.833, -37.968, 91.172, -136.154, 62.336, 156.864]
  MoveL 6739 to (-246.51, 302.72, -54.5) mm, rotated rx 180 ry 0 rz 0.01 deg; joints [37.738, -38.028, 91.303, -136.278, 62.349, 156.967]
  MoveL 6740 to (-246.55, 302.54, -54.5) mm, rotated rx 180 ry 0 rz 0.01 deg; joints [37.732, -38.031, 91.312, -136.285, 62.35, 156.973]
  MoveL 6741 to (-247.04, 299.63, -54.5) mm, rotated rx 180 ry 0 rz 0.01 deg; joints [37.641, -38.097, 91.456, -136.408, 62.369, 157.079]
  MoveL 6742 to (-247.07, 299.4, -54.5) mm, rotated rx -180 ry 0 rz 0.01 deg; joints [37.634, -38.103, 91.468, -136.417, 62.371, 157.088]
  MoveL 6743 to (-260.63, 163.73, -54.5) mm, rotated rx 180 ry 0 rz 0.01 deg; joints [33.371, -41.183, 98.291, -142.105, 63.619, 161.894]
  MoveL 6744 to (-260.63, 163.13, -54.5) mm, rotated rx 180 ry 0 rz 0.01 deg; joints [33.353, -41.198, 98.323, -142.13, 63.626, 161.915]
  MoveL 6745 to (-260.49, 161.32, -54.5) mm, rotated rx -180 ry 0 rz 0.01 deg; joints [33.3, -41.247, 98.431, -142.204, 63.656, 161.981]
  MoveL 6746 to (-260.36, 160.61, -54.5) mm, rotated rx 180 ry 0 rz 0.01 deg; joints [33.281, -41.268, 98.48, -142.232, 63.671, 162.008]
  MoveL 6747 to (-260.03, 159.53, -54.5) mm, rotated rx -180 ry 0 rz 0.01 deg; joints [33.254, -41.307, 98.564, -142.274, 63.698, 162.053]
  MoveL 6748 to (-259.87, 159.09, -54.5) mm, rotated rx -180 ry 0 rz 0.01 deg; joints [33.244, -41.324, 98.601, -142.291, 63.711, 162.072]
  MoveL 6749 to (-259.33, 157.91, -54.5) mm, rotated rx 180 ry 0 rz 0.01 deg; joints [33.218, -41.372, 98.708, -142.335, 63.749, 162.123]
  MoveL 6750 to (-259.03, 157.39, -54.5) mm, rotated rx -180 ry 0 rz 0.01 deg; joints [33.208, -41.396, 98.76, -142.355, 63.768, 162.148]
  MoveL 6751 to (-257.75, 155.55, -54.5) mm, rotated rx 180 ry 0 rz 0.01 deg; joints [33.177, -41.488, 98.962, -142.42, 63.845, 162.237]
  MoveL 6752 to (-257.46, 155.19, -54.5) mm, rotated rx 180 ry 0 rz 0.01 deg; joints [33.172, -41.507, 99.004, -142.433, 63.861, 162.255]
  MoveL 6753 to (-255.84, 153.43, -54.5) mm, rotated rx -180 ry 0 rz 0.01 deg; joints [33.15, -41.609, 99.229, -142.492, 63.951, 162.348]
  MoveL 6754 to (-255.53, 153.13, -54.5) mm, rotated rx -180 ry 0 rz 0.01 deg; joints [33.147, -41.628, 99.27, -142.502, 63.968, 162.365]
  MoveL 6755 to (-253.46, 151.38, -54.5) mm, rotated rx -180 ry 0 rz 0.01 deg; joints [33.135, -41.747, 99.53, -142.557, 64.076, 162.466]
  MoveL 6756 to (-253.22, 151.2, -54.5) mm, rotated rx 180 ry 0 rz 0.01 deg; joints [33.134, -41.76, 99.558, -142.562, 64.088, 162.477]
  MoveL 6757 to (-250.95, 149.6, -54.5) mm, rotated rx -180 ry 0 rz 0.01 deg; joints [33.13, -41.883, 99.827, -142.609, 64.202, 162.577]
  MoveL 6758 to (-250.69, 149.43, -54.5) mm, rotated rx 180 ry 0 rz 0.01 deg; joints [33.131, -41.896, 99.856, -142.613, 64.215, 162.588]
  MoveL 6759 to (-214.41, 128.45, -54.5) mm, rotated rx 180 ry 0 rz 0.01 deg; joints [33.217, -43.701, 103.816, -143.127, 65.96, 163.983]
  MoveC 6760 to (-213.96, 128.23, -54.5) mm, rotated rx 180 ry 0 rz 0.01 deg; joints [33.219, -43.722, 103.863, -143.131, 65.981, 163.999] to (-213.47, 128.08, -54.5) mm, rotated rx 180 ry 0 rz 0.01 deg; joints [33.225, -43.743, 103.908, -143.132, 66.003, 164.012]
  MoveL 6761 to (-212.38, 127.84, -54.5) mm, rotated rx 180 ry 0 rz 0.01 deg; joints [33.24, -43.787, 104.006, -143.131, 66.049, 164.041]
  MoveC 6762 to (-211.85, 127.76, -54.5) mm, rotated rx 180 ry 0 rz 0.01 deg; joints [33.248, -43.808, 104.051, -143.128, 66.072, 164.053] to (-211.31, 127.77, -54.5) mm, rotated rx 180 ry 0 rz 0.01 deg; joints [33.26, -43.827, 104.093, -143.122, 66.093, 164.063]
  MoveL 6763 to (-210.22, 127.87, -54.5) mm, rotated rx -180 ry 0 rz 0.01 deg; joints [33.286, -43.864, 104.172, -143.106, 66.135, 164.08]
  MoveC 6764 to (-209.68, 127.97, -54.5) mm, rotated rx 180 ry 0 rz 0.01 deg; joints [33.301, -43.881, 104.209, -143.096, 66.155, 164.087] to (-209.17, 128.15, -54.5) mm, rotated rx 180 ry 0 rz 0.01 deg; joints [33.317, -43.895, 104.239, -143.084, 66.174, 164.09]
  MoveL 6765 to (-208.14, 128.6, -54.5) mm, rotated rx 180 ry 0 rz 0.01 deg; joints [33.354, -43.921, 104.296, -143.054, 66.209, 164.094]
  MoveL 6766 to (-207.32, 129.12, -54.5) mm, rotated rx -180 ry 0 rz 0.01 deg; joints [33.387, -43.939, 104.333, -143.023, 66.235, 164.093]
  MoveL 6767 to (-206.66, 129.68, -54.5) mm, rotated rx 180 ry 0 rz 0.01 deg; joints [33.419, -43.949, 104.356, -142.993, 66.253, 164.087]
  MoveL 6768 to (-206.04, 130.37, -54.5) mm, rotated rx 180 ry 0 rz 0.01 deg; joints [33.454, -43.956, 104.368, -142.958, 66.269, 164.076]
  MoveL 6769 to (-205.46, 131.24, -54.5) mm, rotated rx -180 ry 0 rz 0.01 deg; joints [33.494, -43.957, 104.369, -142.917, 66.28, 164.058]
  MoveL 6770 to (-205.05, 132.11, -54.5) mm, rotated rx -180 ry 0 rz 0.01 deg; joints [33.531, -43.952, 104.357, -142.876, 66.285, 164.038]
  MoveL 6771 to (-204.77, 133, -54.5) mm, rotated rx 180 ry 0 rz 0.01 deg; joints [33.566, -43.941, 104.332, -142.837, 66.285, 164.013]
  MoveC 6772 to (-204.65, 133.5, -54.5) mm, rotated rx 180 ry 0 rz 0.01 deg; joints [33.584, -43.934, 104.316, -142.815, 66.283, 163.999] to (-204.61, 134.02, -54.5) mm, rotated rx 180 ry 0 rz 0.01 deg; joints [33.601, -43.924, 104.293, -142.793, 66.277, 163.983]
  MoveL 6773 to (-204.67, 267.36, -54.5) mm, rotated rx 180 ry 0 rz 0.01 deg; joints [37.653, -40.599, 96.861, -137.388, 64.493, 159.291]
  MoveL 6774 to (-188.85, 267.36, -54.5) mm, rotated rx 180 ry 0 rz 0.01 deg; joints [38.008, -41.171, 98.09, -137.234, 65.109, 159.625]
  MoveL 6775 to (-188.9, 134.02, -54.5) mm, rotated rx -180 ry 0 rz 0.01 deg; joints [33.938, -44.475, 105.498, -142.615, 66.898, 164.273]
  MoveC 6776 to (-188.86, 133.5, -54.5) mm, rotated rx 180 ry 0 rz 0.01 deg; joints [33.922, -44.488, 105.527, -142.636, 66.906, 164.29] to (-188.75, 133, -54.5) mm, rotated rx 180 ry 0 rz 0.01 deg; joints [33.909, -44.503, 105.562, -142.655, 66.917, 164.308]
  MoveL 6777 to (-188.47, 132.11, -54.5) mm, rotated rx -180 ry 0 rz 0.01 deg; joints [33.886, -44.533, 105.629, -142.688, 66.94, 164.343]
  MoveL 6778 to (-188.05, 131.24, -54.5) mm, rotated rx 180 ry 0 rz 0.01 deg; joints [33.867, -44.567, 105.705, -142.719, 66.969, 164.378]
  MoveL 6779 to (-187.47, 130.37, -54.5) mm, rotated rx -180 ry 0 rz 0.01 deg; joints [33.852, -44.607, 105.794, -142.747, 67.003, 164.417]
  MoveL 6780 to (-186.85, 129.68, -54.5) mm, rotated rx -180 ry 0 rz 0.01 deg; joints [33.843, -44.644, 105.876, -142.768, 67.036, 164.45]
  MoveL 6781 to (-186.2, 129.12, -54.5) mm, rotated rx -180 ry 0 rz 0.01 deg; joints [33.839, -44.679, 105.954, -142.783, 67.069, 164.48]
  MoveL 6782 to (-185.37, 128.6, -54.5) mm, rotated rx 180 ry 0 rz 0.01 deg; joints [33.84, -44.719, 106.043, -142.794, 67.109, 164.512]
  MoveL 6783 to (-184.34, 128.15, -54.5) mm, rotated rx -180 ry 0 rz 0.01 deg; joints [33.847, -44.765, 106.145, -142.801, 67.155, 164.545]
  MoveC 6784 to (-183.83, 127.97, -54.5) mm, rotated rx 180 ry 0 rz 0.01 deg; joints [33.853, -44.787, 106.193, -142.802, 67.178, 164.56] to (-183.29, 127.87, -54.5) mm, rotated rx 180 ry 0 rz 0.01 deg; joints [33.861, -44.807, 106.238, -142.799, 67.2, 164.573]
  MoveL 6785 to (-182.2, 127.77, -54.5) mm, rotated rx 180 ry 0 rz 0.01 deg; joints [33.881, -44.847, 106.326, -142.79, 67.244, 164.596]
  MoveC 6786 to (-181.66, 127.76, -54.5) mm, rotated rx -180 ry 0 rz 0.01 deg; joints [33.893, -44.866, 106.367, -142.784, 67.265, 164.606] to (-181.13, 127.84, -54.5) mm, rotated rx -180 ry 0 rz 0.01 deg; joints [33.907, -44.883, 106.404, -142.775, 67.285, 164.613]
  MoveL 6787 to (-180.04, 128.08, -54.5) mm, rotated rx 180 ry 0 rz 0.01 deg; joints [33.939, -44.915, 106.474, -142.751, 67.324, 164.625]
  MoveC 6788 to (-179.56, 128.23, -54.5) mm, rotated rx 180 ry 0 rz 0.01 deg; joints [33.954, -44.928, 106.503, -142.739, 67.341, 164.629] to (-179.1, 128.45, -54.5) mm, rotated rx -180 ry 0 rz 0.01 deg; joints [33.971, -44.939, 106.526, -142.725, 67.356, 164.63]
  MoveL 6789 to (-142.82, 149.43, -54.5) mm, rotated rx -180 ry 0 rz 0.01 deg; joints [35.458, -45.693, 108.147, -141.404, 68.469, 164.611]
  MoveL 6790 to (-142.61, 149.57, -54.5) mm, rotated rx -180 ry 0 rz 0.01 deg; joints [35.467, -45.697, 108.155, -141.396, 68.475, 164.611]
  MoveL 6791 to (-141.16, 150.55, -54.5) mm, rotated rx 180 ry 0 rz 0.01 deg; joints [35.532, -45.723, 108.21, -141.336, 68.516, 164.605]
  MoveL 6792 to (-140.93, 150.73, -54.5) mm, rotated rx -180 ry 0 rz 0.01 deg; joints [35.543, -45.726, 108.218, -141.326, 68.523, 164.604]
  MoveL 6793 to (-138.02, 153.1, -54.5) mm, rotated rx 180 ry 0 rz 0.01 deg; joints [35.686, -45.769, 108.307, -141.191, 68.6, 164.58]
  MoveL 6794 to (-137.73, 153.36, -54.5) mm, rotated rx 180 ry 0 rz 0.01 deg; joints [35.701, -45.772, 108.314, -141.176, 68.607, 164.576]
  MoveL 6795 to (-136.62, 154.52, -54.5) mm, rotated rx 180 ry 0 rz 0.01 deg; joints [35.764, -45.783, 108.335, -141.114, 68.634, 164.559]
  MoveL 6796 to (-136.37, 154.8, -54.5) mm, rotated rx -180 ry 0 rz 0.01 deg; joints [35.779, -45.784, 108.338, -141.099, 68.639, 164.555]
  MoveL 6797 to (-134.95, 156.64, -54.5) mm, rotated rx 180 ry 0 rz 0.01 deg; joints [35.871, -45.789, 108.345, -141.005, 68.668, 164.521]
  MoveL 6798 to (-134.65, 157.1, -54.5) mm, rotated rx -180 ry 0 rz 0.01 deg; joints [35.893, -45.788, 108.343, -140.982, 68.672, 164.511]
  MoveL 6799 to (-133.88, 158.53, -54.5) mm, rotated rx -180 ry 0 rz 0.01 deg; joints [35.956, -45.781, 108.324, -140.914, 68.682, 164.479]
  MoveL 6800 to (-133.63, 159.11, -54.5) mm, rotated rx 180 ry 0 rz 0.01 deg; joints [35.98, -45.776, 108.311, -140.888, 68.683, 164.465]
  MoveL 6801 to (-133.17, 160.56, -54.5) mm, rotated rx 180 ry 0 rz 0.01 deg; joints [36.037, -45.757, 108.268, -140.823, 68.681, 164.426]
  MoveL 6802 to (-133.02, 161.32, -54.5) mm, rotated rx -180 ry 0 rz 0.01 deg; joints [36.065, -45.745, 108.239, -140.79, 68.676, 164.404]
  MoveL 6803 to (-132.88, 163.13, -54.5) mm, rotated rx 180 ry 0 rz 0.01 deg; joints [36.126, -45.707, 108.153, -140.716, 68.656, 164.348]
  MoveL 6804 to (-132.88, 163.73, -54.5) mm, rotated rx 180 ry 0 rz 0.01 deg; joints [36.145, -45.693, 108.121, -140.692, 68.648, 164.328]
  MoveL 6805 to (-145.51, 290.23, -54.5) mm, rotated rx -180 ry 0 rz 0.01 deg; joints [39.672, -42.061, 99.976, -135.847, 66.448, 159.663]
  MoveL 6806 to (-146.65, 300.88, -54.5) mm, rotated rx 180 ry 0 rz 0.01 deg; joints [39.948, -41.726, 99.235, -135.443, 66.261, 159.238]
  MoveL 6807 to (-146.7, 301.22, -54.5) mm, rotated rx 180 ry 0 rz 0.01 deg; joints [39.957, -41.714, 99.209, -135.43, 66.254, 159.223]
  MoveL 6808 to (-147.48, 304.85, -54.5) mm, rotated rx -180 ry 0 rz 0.01 deg; joints [40.041, -41.585, 98.926, -135.296, 66.176, 159.069]
  MoveL 6809 to (-147.54, 305.09, -54.5) mm, rotated rx 180 ry 0 rz 0.01 deg; joints [40.047, -41.576, 98.906, -135.288, 66.171, 159.059]
  MoveL 6810 to (-148.33, 307.82, -54.5) mm, rotated rx 180 ry 0 rz 0.01 deg; joints [40.105, -41.472, 98.677, -135.19, 66.104, 158.938]
  MoveL 6811 to (-148.5, 308.73, -54.5) mm, rotated rx -180 ry 0 rz 0.01 deg; joints [40.127, -41.44, 98.607, -135.156, 66.086, 158.9]
  MoveL 6812 to (-148.64, 309.28, -54.5) mm, rotated rx 180 ry 0 rz 0.01 deg; joints [40.139, -41.42, 98.562, -135.136, 66.073, 158.876]
  MoveL 6813 to (-149.56, 311.82, -54.5) mm, rotated rx -180 ry 0 rz 0.01 deg; joints [40.188, -41.316, 98.335, -135.047, 66.004, 158.759]
  MoveL 6814 to (-149.79, 312.34, -54.5) mm, rotated rx -180 ry 0 rz 0.01 deg; joints [40.197, -41.293, 98.284, -135.029, 65.988, 158.734]
  MoveL 6815 to (-155.12, 321.77, -54.5) mm, rotated rx 180 ry 0 rz 0.01 deg; joints [40.335, -40.837, 97.288, -134.719, 65.66, 158.256]
  MoveL 6816 to (-155.42, 322.2, -54.5) mm, rotated rx 180 ry 0 rz 0.01 deg; joints [40.34, -40.814, 97.238, -134.705, 65.643, 158.233]
  MoveL 6817 to (-156.85, 324.02, -54.5) mm, rotated rx 180 ry 0 rz 0.01 deg; joints [40.357, -40.711, 97.014, -134.649, 65.565, 158.131]
  MoveL 6818 to (-157.19, 324.39, -54.5) mm, rotated rx -180 ry 0 rz 0.01 deg; joints [40.359, -40.689, 96.965, -134.638, 65.547, 158.11]
  MoveL 6819 to (-165.06, 331.76, -54.5) mm, rotated rx 180 ry 0 rz 0.01 deg; joints [40.378, -40.196, 95.896, -134.43, 65.15, 157.649]
  MoveL 6820 to (-165.37, 332.01, -54.5) mm, rotated rx -180 ry 0 rz 0.01 deg; joints [40.378, -40.178, 95.856, -134.423, 65.135, 157.632]
  MoveL 6821 to (-166.82, 333.08, -54.5) mm, rotated rx 180 ry 0 rz 0.01 deg; joints [40.373, -40.095, 95.676, -134.396, 65.066, 157.558]
  MoveL 6822 to (-167.35, 333.4, -54.5) mm, rotated rx -180 ry 0 rz 0.01 deg; joints [40.369, -40.067, 95.616, -134.389, 65.041, 157.534]
  MoveL 6823 to (-177.87, 338.5, -54.5) mm, rotated rx -180 ry 0 rz 0.01 deg; joints [40.264, -39.538, 94.476, -134.289, 64.571, 157.097]
  MoveL 6824 to (-178.25, 338.66, -54.5) mm, rotated rx -180 ry 0 rz 0.01 deg; joints [40.26, -39.52, 94.436, -134.287, 64.555, 157.082]
  MoveL 6825 to (-179.34, 339.03, -54.5) mm, rotated rx 180 ry 0 rz 0.01 deg; joints [40.245, -39.469, 94.327, -134.282, 64.508, 157.043]
  MoveL 6826 to (-179.93, 339.17, -54.5) mm, rotated rx -180 ry 0 rz 0.01 deg; joints [40.235, -39.444, 94.273, -134.282, 64.483, 157.024]
  MoveL 6827 to (-180.14, 339.2, -54.5) mm, rotated rx -180 ry 0 rz 0.01 deg; joints [40.231, -39.435, 94.254, -134.283, 64.475, 157.018]
  MoveL 6828 to (4.87, 339.21, -54.5) mm, rotated rx -180 ry 0 rz 0.01 deg; joints [44.922, -45.451, 107.29, -131.695, 71.063, 160.745]
  MoveL 6829 to (5.94, 339.15, -54.5) mm, rotated rx -180 ry 0 rz 0.01 deg; joints [44.95, -45.484, 107.363, -131.677, 71.099, 160.767]
  MoveL 6830 to (6.8, 338.95, -54.5) mm, rotated rx -180 ry 0 rz 0.01 deg; joints [44.968, -45.515, 107.431, -131.668, 71.13, 160.79]
  MoveL 6831 to (7.07, 338.84, -54.5) mm, rotated rx -180 ry 0 rz 0.01 deg; joints [44.972, -45.526, 107.455, -131.668, 71.141, 160.799]
  MoveL 6832 to (7.57, 338.46, -54.33) mm, rotated rx 180 ry 0 rz 0.01 deg; joints [44.975, -45.56, 107.513, -131.671, 71.157, 160.816]
  MoveL 6833 to (7.78, 338.05, -53.87) mm, rotated rx 180 ry 0 rz 0.01 deg; joints [44.97, -45.604, 107.555, -131.676, 71.155, 160.818]
  MoveL 6834 to (7.82, 337.88, -53.23) mm, rotated rx -180 ry 0 rz 0.01 deg; joints [44.966, -45.644, 107.572, -131.674, 71.138, 160.8]
  Set speed (1000.0 mm/s)
  MoveL 6835 to (7.82, 337.88, 11) mm, rotated rx 180 ry 0 rz 0.01 deg; joints [44.942, -49.073, 107.797, -130.824, 69.015, 158.246]
  Set speed (1000.0 mm/s)
  MoveL 6836 to (-66.82, 254.06, 11) mm, rotated rx -180 ry 0 rz 0.01 deg; joints [40.524, -49.102, 107.981, -135.273, 67.449, 160.05]
  Set speed (1000.0 mm/s)
  MoveL 6837 to (-66.82, 254.06, -42.73) mm, rotated rx 180 ry 0 rz 0.01 deg; joints [40.548, -46.238, 107.815, -135.995, 69.387, 162.07]
  Set speed (100.0 mm/s)
  MoveL 6838 to (-66.66, 254.05, -43.35) mm, rotated rx 180 ry 0 rz 0.01 deg; joints [40.552, -46.21, 107.824, -136.001, 69.415, 162.096]
  MoveL 6839 to (-66.21, 254.02, -43.82) mm, rotated rx -180 ry 0 rz 0.01 deg; joints [40.563, -46.199, 107.854, -136, 69.447, 162.122]
  MoveL 6840 to (-65.6, 254.03, -44) mm, rotated rx -180 ry 0 rz 0.01 deg; joints [40.579, -46.208, 107.894, -135.992, 69.475, 162.139]
  MoveL 6841 to (-60.36, 258.06, -44.24) mm, rotated rx -180 ry 0 rz 0.01 deg; joints [40.834, -46.254, 108.014, -135.755, 69.612, 162.102]
  MoveL 6842 to (-61.95, 264.47, -44.49) mm, rotated rx -180 ry 0 rz 0.01 deg; joints [40.983, -46.022, 107.526, -135.537, 69.479, 161.856]
  MoveL 6843 to (-68.46, 265.58, -44.73) mm, rotated rx 180 ry 0 rz 0.01 deg; joints [40.849, -45.774, 107.013, -135.602, 69.244, 161.707]
  MoveL 6844 to (-72.09, 260.06, -44.98) mm, rotated rx -180 ry 0 rz 0.01 deg; joints [40.593, -45.792, 107.088, -135.875, 69.2, 161.844]
  MoveL 6845 to (-68.49, 254.53, -45.22) mm, rotated rx 180 ry 0 rz 0.01 deg; joints [40.52, -46.038, 107.66, -136.035, 69.41, 162.113]
  MoveL 6846 to (-61.97, 255.61, -45.46) mm, rotated rx 180 ry 0 rz 0.01 deg; joints [40.72, -46.201, 108.042, -135.89, 69.632, 162.203]
  MoveL 6847 to (-60.35, 262.01, -45.71) mm, rotated rx -180 ry 0 rz 0.01 deg; joints [40.952, -46.071, 107.774, -135.62, 69.611, 162.016]
  MoveL 6848 to (-65.57, 266.06, -45.95) mm, rotated rx 180 ry 0 rz 0.01 deg; joints [40.938, -45.787, 107.176, -135.552, 69.382, 161.787]
  MoveL 6849 to (-71.37, 262.9, -46.2) mm, rotated rx 180 ry 0 rz 0.01 deg; joints [40.696, -45.674, 106.963, -135.769, 69.229, 161.801]
  MoveL 6850 to (-70.8, 256.32, -46.44) mm, rotated rx 180 ry 0 rz 0.01 deg; joints [40.515, -45.852, 107.389, -136.017, 69.347, 162.052]
  MoveL 6851 to (-64.55, 254.21, -46.68) mm, rotated rx 180 ry 0 rz 0.01 deg; joints [40.612, -46.091, 107.941, -136.001, 69.604, 162.249]
  MoveL 6852 to (-60.1, 259.09, -46.93) mm, rotated rx -180 ry 0 rz 0.01 deg; joints [40.872, -46.089, 107.957, -135.743, 69.702, 162.168]
  MoveL 6853 to (-62.79, 265.12, -47.17) mm, rotated rx -180 ry 0 rz 0.01 deg; joints [40.982, -45.833, 107.415, -135.559, 69.534, 161.915]
  MoveL 6854 to (-69.4, 265.07, -47.42) mm, rotated rx 180 ry 0 rz 0.01 deg; joints [40.812, -45.613, 106.964, -135.67, 69.312, 161.804]
  MoveL 6855 to (-72, 259, -47.66) mm, rotated rx 180 ry 0 rz 0.01 deg; joints [40.565, -45.678, 107.142, -135.948, 69.311, 161.979]
  MoveL 6856 to (-67.48, 254.18, -47.9) mm, rotated rx 180 ry 0 rz 0.01 deg; joints [40.537, -45.933, 107.735, -136.064, 69.545, 162.24]
  MoveL 6857 to (-61.25, 256.4, -48.15) mm, rotated rx -180 ry 0 rz 0.01 deg; joints [40.763, -46.057, 108.029, -135.881, 69.741, 162.285]
  MoveL 6858 to (-60.79, 262.98, -48.39) mm, rotated rx 180 ry 0 rz 0.01 deg; joints [40.971, -45.885, 107.671, -135.623, 69.676, 162.071]
  MoveL 6859 to (-66.64, 266.05, -48.64) mm, rotated rx -180 ry 0 rz 0.01 deg; joints [40.912, -45.608, 107.088, -135.603, 69.438, 161.864]
  MoveL 6860 to (-71.79, 261.92, -48.88) mm, rotated rx -180 ry 0 rz 0.01 deg; joints [40.658, -45.541, 106.977, -135.847, 69.321, 161.924]
  MoveL 6861 to (-70.07, 255.55, -49.13) mm, rotated rx -180 ry 0 rz 0.01 deg; joints [40.512, -45.749, 107.469, -136.068, 69.477, 162.189]
  MoveL 6862 to (-63.54, 254.56, -49.37) mm, rotated rx 180 ry 0 rz 0.01 deg; joints [40.65, -45.966, 107.974, -136.004, 69.729, 162.351]
  MoveL 6863 to (-60.02, 260.15, -49.61) mm, rotated rx 180 ry 0 rz 0.01 deg; joints [40.907, -45.917, 107.884, -135.734, 69.784, 162.229]
  MoveL 6864 to (-63.74, 265.62, -49.86) mm, rotated rx 180 ry 0 rz 0.01 deg; joints [40.974, -45.644, 107.305, -135.588, 69.588, 161.977]
  MoveL 6865 to (-70.23, 264.4, -50.1) mm, rotated rx -180 ry 0 rz 0.01 deg; joints [40.772, -45.459, 106.93, -135.742, 69.385, 161.909]
  MoveL 6866 to (-71.72, 257.97, -50.35) mm, rotated rx 180 ry 0 rz 0.01 deg; joints [40.543, -45.568, 107.206, -136.016, 69.429, 162.117]
  MoveL 6867 to (-66.42, 254.03, -50.59) mm, rotated rx 180 ry 0 rz 0.01 deg; joints [40.56, -45.824, 107.801, -136.086, 69.678, 162.361]
  MoveL 6868 to (-60.69, 257.3, -50.83) mm, rotated rx -180 ry 0 rz 0.01 deg; joints [40.806, -45.904, 107.999, -135.869, 69.843, 162.361]
  MoveL 6869 to (-61.39, 263.87, -51.08) mm, rotated rx -180 ry 0 rz 0.01 deg; joints [40.983, -45.697, 107.563, -135.631, 69.737, 162.126]
  MoveL 6870 to (-67.68, 265.86, -51.32) mm, rotated rx 180 ry 0 rz 0.01 deg; joints [40.88, -45.435, 107.012, -135.66, 69.497, 161.948]
  MoveL 6871 to (-72.03, 260.88, -51.57) mm, rotated rx -180 ry 0 rz 0.01 deg; joints [40.622, -45.416, 107.006, -135.924, 69.42, 162.052]
  MoveL 6872 to (-69.22, 254.91, -51.81) mm, rotated rx -180 ry 0 rz 0.01 deg; joints [40.516, -45.647, 107.55, -136.112, 69.611, 162.323]
  MoveL 6873 to (-62.61, 255.09, -52.05) mm, rotated rx 180 ry 0 rz 0.01 deg; joints [40.691, -45.835, 107.99, -136, 69.849, 162.446]
  MoveL 6874 to (-60.14, 261.22, -52.3) mm, rotated rx 180 ry 0 rz 0.01 deg; joints [40.937, -45.739, 107.797, -135.727, 69.86, 162.286]
  MoveL 6875 to (-64.75, 265.94, -52.54) mm, rotated rx -180 ry 0 rz 0.01 deg; joints [40.958, -45.458, 107.201, -135.624, 69.641, 162.043]
  MoveL 6876 to (-70.93, 263.6, -52.79) mm, rotated rx 180 ry 0 rz 0.01 deg; joints [40.731, -45.313, 106.914, -135.816, 69.464, 162.02]
  MoveL 6877 to (-71.27, 257, -53.03) mm, rotated rx -180 ry 0 rz 0.01 deg; joints [40.527, -45.462, 107.278, -136.078, 69.552, 162.255]
  MoveL 6878 to (-65.36, 254.06, -53.27) mm, rotated rx -180 ry 0 rz 0.01 deg; joints [40.59, -45.71, 107.856, -136.1, 69.81, 162.476]
  MoveL 6879 to (-60.29, 258.29, -53.52) mm, rotated rx -180 ry 0 rz 0.01 deg; joints [40.847, -45.744, 107.952, -135.857, 69.938, 162.43]
  MoveL 6880 to (-62.13, 264.63, -53.76) mm, rotated rx 180 ry 0 rz 0.01 deg; joints [40.988, -45.508, 107.45, -135.647, 69.793, 162.182]
  MoveL 6881 to (-68.68, 265.48, -54.01) mm, rotated rx 180 ry 0 rz 0.01 deg; joints [40.845, -45.268, 106.95, -135.723, 69.56, 162.039]
  MoveL 6882 to (-72.08, 259.82, -54.25) mm, rotated rx 180 ry 0 rz 0.01 deg; joints [40.59, -45.296, 107.049, -135.998, 69.526, 162.184]
  MoveL 6883 to (-68.26, 254.43, -54.49) mm, rotated rx 180 ry 0 rz 0.01 deg; joints [40.527, -45.543, 107.627, -136.147, 69.745, 162.452]
  MoveL 6884 to (-61.8, 255.78, -54.74) mm, rotated rx 180 ry 0 rz 0.01 deg; joints [40.733, -45.695, 107.989, -135.993, 69.963, 162.534]
  MoveL 6885 to (-60.44, 262.24, -54.98) mm, rotated rx 180 ry 0 rz 0.01 deg; joints [40.961, -45.556, 107.7, -135.725, 69.929, 162.341]
  MoveL 6886 to (-65.81, 266.07, -55.23) mm, rotated rx 180 ry 0 rz 0.01 deg; joints [40.936, -45.276, 107.104, -135.669, 69.695, 162.115]
  MoveL 6887 to (-71.48, 262.69, -55.47) mm, rotated rx -180 ry 0 rz 0.01 deg; joints [40.691, -45.174, 106.913, -135.893, 69.55, 162.138]
  MoveL 6888 to (-70.65, 256.13, -55.71) mm, rotated rx 180 ry 0 rz 0.01 deg; joints [40.518, -45.357, 107.355, -136.134, 69.68, 162.392]
  MoveL 6889 to (-64.31, 254.27, -55.96) mm, rotated rx -180 ry 0 rz 0.01 deg; joints [40.624, -45.589, 107.898, -136.106, 69.938, 162.583]
  MoveL 6890 to (-60.07, 259.33, -56.2) mm, rotated rx 180 ry 0 rz 0.01 deg; joints [40.885, -45.577, 107.889, -135.845, 70.025, 162.494]
  MoveL 6891 to (-63, 265.25, -56.45) mm, rotated rx 180 ry 0 rz 0.01 deg; joints [40.985, -45.318, 107.337, -135.669, 69.847, 162.24]
  MoveL 6892 to (-69.6, 264.93, -56.69) mm, rotated rx -180 ry 0 rz 0.01 deg; joints [40.806, -45.108, 106.902, -135.791, 69.628, 162.137]
  MoveL 6893 to (-71.95, 258.76, -56.93) mm, rotated rx -180 ry 0 rz 0.01 deg; joints [40.563, -45.182, 107.103, -136.069, 69.639, 162.319]
  MoveL 6894 to (-67.24, 254.13, -57.18) mm, rotated rx 180 ry 0 rz 0.01 deg; joints [40.546, -45.435, 107.698, -136.174, 69.879, 162.577]
  MoveL 6895 to (-61.11, 256.59, -57.42) mm, rotated rx -180 ry 0 rz 0.01 deg; joints [40.777, -45.548, 107.971, -135.982, 70.069, 162.614]
  MoveL 6896 to (-60.91, 263.19, -57.67) mm, rotated rx -180 ry 0 rz 0.01 deg; joints [40.978, -45.37, 107.594, -135.728, 69.992, 162.395]
  MoveL 6897 to (-66.88, 266.02, -57.91) mm, rotated rx 180 ry 0 rz 0.01 deg; joints [40.909, -45.098, 107.016, -135.72, 69.75, 162.192]
  MoveL 6898 to (-71.86, 261.69, -58.15) mm, rotated rx -180 ry 0 rz 0.01 deg; joints [40.653, -45.042, 106.929, -135.969, 69.643, 162.261]
  MoveL 6899 to (-69.89, 255.39, -58.4) mm, rotated rx -180 ry 0 rz 0.01 deg; joints [40.516, -45.254, 107.434, -136.183, 69.811, 162.527]
  MoveL 6900 to (-63.32, 254.67, -58.64) mm, rotated rx -180 ry 0 rz 0.01 deg; joints [40.663, -45.463, 107.925, -136.106, 70.061, 162.683]
  MoveL 6901 to (-60.03, 260.4, -58.89) mm, rotated rx -180 ry 0 rz 0.01 deg; joints [40.918, -45.403, 107.811, -135.835, 70.104, 162.553]
  MoveL 6902 to (-63.96, 265.71, -59.13) mm, rotated rx -180 ry 0 rz 0.01 deg; joints [40.975, -45.13, 107.227, -135.699, 69.899, 162.301]
  MoveL 6903 to (-70.4, 264.23, -59.37) mm, rotated rx -180 ry 0 rz 0.01 deg; joints [40.766, -44.955, 106.871, -135.863, 69.701, 162.241]
  MoveL 6904 to (-71.63, 257.74, -59.62) mm, rotated rx -180 ry 0 rz 0.01 deg; joints [40.542, -45.072, 107.168, -136.134, 69.758, 162.455]
  MoveL 6905 to (-66.18, 254.02, -59.86) mm, rotated rx 180 ry 0 rz 0.01 deg; joints [40.571, -45.324, 107.76, -136.192, 70.012, 162.696]
  MoveL 6906 to (-60.58, 257.52, -60.11) mm, rotated rx 180 ry 0 rz 0.01 deg; joints [40.819, -45.393, 107.935, -135.969, 70.168, 162.687]
  MoveL 6907 to (-61.55, 264.05, -60.35) mm, rotated rx -180 ry 0 rz 0.01 deg; joints [40.989, -45.181, 107.482, -135.737, 70.05, 162.448]
  MoveL 6908 to (-67.92, 265.79, -60.6) mm, rotated rx 180 ry 0 rz 0.01 deg; joints [40.876, -44.926, 106.941, -135.778, 69.809, 162.276]
  MoveL 6909 to (-72.06, 260.64, -60.84) mm, rotated rx -180 ry 0 rz 0.01 deg; joints [40.618, -44.917, 106.959, -136.044, 69.744, 162.388]
  MoveL 6910 to (-69.01, 254.79, -61.08) mm, rotated rx 180 ry 0 rz 0.01 deg; joints [40.522, -45.15, 107.512, -136.223, 69.944, 162.659]
  MoveL 6911 to (-62.42, 255.24, -61.33) mm, rotated rx 180 ry 0 rz 0.01 deg; joints [40.704, -45.328, 107.936, -136.101, 70.179, 162.775]
  MoveL 6912 to (-60.19, 261.45, -61.57) mm, rotated rx 180 ry 0 rz 0.01 deg; joints [40.947, -45.223, 107.72, -135.829, 70.177, 162.608]
  MoveL 6913 to (-64.99, 265.99, -61.82) mm, rotated rx -180 ry 0 rz 0.01 deg; joints [40.958, -44.944, 107.122, -135.737, 69.952, 162.367]
  MoveL 6914 to (-71.07, 263.4, -62.06) mm, rotated rx -180 ry 0 rz 0.01 deg; joints [40.726, -44.81, 106.856, -135.937, 69.782, 162.353]
  MoveL 6915 to (-71.14, 256.8, -62.3) mm, rotated rx -180 ry 0 rz 0.01 deg; joints [40.528, -44.965, 107.239, -136.194, 69.882, 162.592]
  MoveL 6916 to (-65.11, 254.09, -62.55) mm, rotated rx -180 ry 0 rz 0.01 deg; joints [40.601, -45.208, 107.81, -136.203, 70.142, 162.808]
  MoveL 6917 to (-60.22, 258.52, -62.79) mm, rotated rx -180 ry 0 rz 0.01 deg; joints [40.859, -45.231, 107.882, -135.955, 70.26, 162.753]
  MoveL 6918 to (-62.32, 264.78, -63.04) mm, rotated rx 180 ry 0 rz 0.01 deg; joints [40.991, -44.991, 107.367, -135.753, 70.105, 162.503]
  MoveL 6919 to (-68.9, 265.37, -63.28) mm, rotated rx 180 ry 0 rz 0.01 deg; joints [40.84, -44.76, 106.88, -135.841, 69.873, 162.367]
  MoveL 6920 to (-72.07, 259.57, -63.52) mm, rotated rx -180 ry 0 rz 0.01 deg; joints [40.587, -44.798, 107.003, -136.117, 69.851, 162.52]
  MoveL 6921 to (-68.03, 254.35, -63.77) mm, rotated rx -180 ry 0 rz 0.01 deg; joints [40.535, -45.044, 107.586, -136.255, 70.078, 162.787]
  MoveL 6922 to (-61.63, 255.95, -64.01) mm, rotated rx -180 ry 0 rz 0.01 deg; joints [40.747, -45.186, 107.929, -136.091, 70.29, 162.86]
  MoveL 6923 to (-60.53, 262.46, -64.26) mm, rotated rx 180 ry 0 rz 0.01 deg; joints [40.969, -45.039, 107.618, -135.827, 70.243, 162.661]
  MoveL 6924 to (-66.06, 266.08, -64.5) mm, rotated rx -180 ry 0 rz 0.01 deg; joints [40.934, -44.763, 107.025, -135.782, 70.005, 162.439]
  MoveL 6925 to (-66.45, 266.08, -64.5) mm, rotated rx -180 ry 0 rz 0.01 deg; joints [40.924, -44.75, 106.998, -135.788, 69.991, 162.431]
  MoveC 6926 to (-68.56, 265.15, -64.5) mm, rotated rx 180 ry 0 rz 0.01 deg; joints [40.843, -44.71, 106.908, -135.858, 69.93, 162.424] to (-69.28, 262.96, -64.5) mm, rotated rx 180 ry 0 rz 0.01 deg; joints [40.76, -44.744, 106.989, -135.954, 69.936, 162.488]
  MoveL 6927 to (-65.15, 221.62, -64.5) mm, rotated rx 180 ry 0 rz 0.01 deg; joints [39.616, -45.911, 109.664, -137.478, 70.678, 163.988]
  MoveC 6928 to (-63.95, 220.59, -64.5) mm, rotated rx 180 ry 0 rz 0.01 deg; joints [39.615, -45.972, 109.804, -137.498, 70.736, 164.045] to (-62.86, 221.74, -64.5) mm, rotated rx -180 ry 0 rz 0.01 deg; joints [39.678, -45.978, 109.814, -137.435, 70.758, 164.026]
  MoveL 6929 to (-62.86, 263.24, -64.5) mm, rotated rx -180 ry 0 rz 0.01 deg; joints [40.932, -44.934, 107.412, -135.838, 70.159, 162.599]
  MoveC 6930 to (-63.69, 265.25, -64.5) mm, rotated rx 180 ry 0 rz 0.01 deg; joints [40.971, -44.857, 107.236, -135.775, 70.1, 162.513] to (-65.7, 266.08, -64.5) mm, rotated rx -180 ry 0 rz 0.01 deg; joints [40.944, -44.774, 107.049, -135.776, 70.018, 162.445]
  MoveL 6931 to (-66.06, 266.08, -64.5) mm, rotated rx -180 ry 0 rz 0.01 deg; joints [40.934, -44.763, 107.025, -135.782, 70.005, 162.439]
  MoveC 6932 to (-68.34, 266.91, -64.5) mm, rotated rx -180 ry 0 rz 0.01 deg; joints [40.901, -44.671, 106.819, -135.787, 69.912, 162.366] to (-69.55, 269.01, -64.5) mm, rotated rx -180 ry 0 rz 0.01 deg; joints [40.932, -44.578, 106.611, -135.726, 69.839, 162.269]
  MoveC 6933 to (-71.23, 271.03, -64.5) mm, rotated rx -180 ry 0 rz 0.01 deg; joints [40.948, -44.474, 106.375, -135.676, 69.751, 162.165] to (-73.82, 270.6, -64.5) mm, rotated rx 180 ry 0 rz 0.01 deg; joints [40.869, -44.404, 106.222, -135.733, 69.665, 162.131]
  MoveC 6934 to (-74.82, 269.26, -64.5) mm, rotated rx -180 ry 0 rz 0.01 deg; joints [40.805, -44.408, 106.233, -135.801, 69.649, 162.16] to (-75.06, 267.61, -64.5) mm, rotated rx -180 ry 0 rz 0.01 deg; joints [40.75, -44.444, 106.314, -135.868, 69.664, 162.214]
  MoveL 6935 to (-66.9, 186, -64.5) mm, rotated rx -180 ry 0 rz 0.01 deg; joints [38.458, -46.707, 111.521, -138.896, 71.134, 165.132]
  MoveC 6936 to (-66.41, 184.48, -64.5) mm, rotated rx 180 ry 0 rz 0.01 deg; joints [38.422, -46.758, 111.638, -138.947, 71.173, 165.191] to (-65.34, 183.29, -64.5) mm, rotated rx 180 ry 0 rz 0.01 deg; joints [38.412, -46.818, 111.776, -138.975, 71.229, 165.248]
  MoveL 6937 to (-60.81, 180.04, -64.5) mm, rotated rx 180 ry 0 rz 0.01 deg; joints [38.422, -47.031, 112.263, -139.025, 71.439, 165.435]
  MoveC 6938 to (-58.68, 179.88, -64.5) mm, rotated rx -180 ry 0 rz 0.01 deg; joints [38.471, -47.098, 112.417, -138.994, 71.518, 165.478] to (-57.57, 181.7, -64.5) mm, rotated rx 180 ry 0 rz 0.01 deg; joints [38.558, -47.09, 112.394, -138.904, 71.531, 165.439]
  MoveL 6939 to (-57.57, 267.52, -64.5) mm, rotated rx -180 ry 0 rz 0.01 deg; joints [41.196, -44.986, 107.519, -135.587, 70.283, 162.548]
  MoveC 6940 to (-58.7, 270.24, -64.5) mm, rotated rx 180 ry 0 rz 0.01 deg; joints [41.247, -44.88, 107.28, -135.502, 70.204, 162.43] to (-61.42, 271.37, -64.5) mm, rotated rx 180 ry 0 rz 0.01 deg; joints [41.21, -44.768, 107.027, -135.504, 70.092, 162.339]
  MoveL 6941 to (-71.65, 271.37, -64.5) mm, rotated rx 180 ry 0 rz 0.01 deg; joints [40.947, -44.451, 106.325, -135.67, 69.731, 162.145]
  MoveC 6942 to (-72.8, 271.17, -64.5) mm, rotated rx -180 ry 0 rz 0.01 deg; joints [40.912, -44.421, 106.258, -135.695, 69.693, 162.13] to (-73.82, 270.6, -64.5) mm, rotated rx -180 ry 0 rz 0.01 deg; joints [40.869, -44.404, 106.222, -135.733, 69.665, 162.131]
  MoveC 6943 to (-76.25, 269.15, -64.5) mm, rotated rx 180 ry 0 rz 0.01 deg; joints [40.765, -44.366, 106.14, -135.827, 69.599, 162.136] to (-79, 268.48, -64.5) mm, rotated rx -180 ry 0 rz 0.01 deg; joints [40.675, -44.298, 105.989, -135.896, 69.511, 162.108]
  MoveC 6944 to (-81.68, 267.05, -64.5) mm, rotated rx 180 ry 0 rz 0.01 deg; joints [40.566, -44.251, 105.888, -135.993, 69.435, 162.107] to (-82.56, 264.15, -64.5) mm, rotated rx -180 ry 0 rz 0.01 deg; joints [40.458, -44.299, 105.999, -136.118, 69.445, 162.194]
  MoveL 6945 to (-74.7, 185.47, -64.5) mm, rotated rx 180 ry 0 rz 0.01 deg; joints [38.246, -46.481, 111.013, -139.048, 70.861, 165.009]
  MoveC 6946 to (-73.13, 180.6, -64.5) mm, rotated rx 180 ry 0 rz 0.01 deg; joints [38.13, -46.642, 111.386, -139.213, 70.988, 165.195] to (-69.7, 176.81, -64.5) mm, rotated rx -180 ry 0 rz 0.01 deg; joints [38.095, -46.835, 111.827, -139.304, 71.167, 165.379]
  MoveL 6947 to (-53, 164.81, -64.5) mm, rotated rx -180 ry 0 rz 0.01 deg; joints [38.13, -47.613, 113.613, -139.487, 71.942, 166.059]
  MoveC 6948 to (-50.87, 164.65, -64.5) mm, rotated rx 180 ry 0 rz 0.01 deg; joints [38.18, -47.68, 113.767, -139.455, 72.021, 166.102] to (-49.75, 166.47, -64.5) mm, rotated rx 180 ry 0 rz 0.01 deg; joints [38.267, -47.672, 113.745, -139.364, 72.033, 166.064]
  MoveL 6949 to (-49.76, 275.33, -64.5) mm, rotated rx 180 ry 0 rz 0.01 deg; joints [41.629, -45.02, 107.582, -135.16, 70.444, 162.418]
  MoveC 6950 to (-50.89, 278.05, -64.5) mm, rotated rx -180 ry 0 rz 0.01 deg; joints [41.679, -44.914, 107.342, -135.075, 70.366, 162.3] to (-53.61, 279.18, -64.5) mm, rotated rx 180 ry 0 rz 0.01 deg; joints [41.641, -44.802, 107.09, -135.078, 70.254, 162.209]
  MoveL 6951 to (-80.28, 279.18, -64.5) mm, rotated rx -180 ry 0 rz 0.01 deg; joints [40.957, -43.976, 105.26, -135.506, 69.312, 161.701]
  MoveC 6952 to (-82.82, 278.06, -64.5) mm, rotated rx 180 ry 0 rz 0.01 deg; joints [40.86, -43.926, 105.151, -135.588, 69.238, 161.692] to (-83.69, 275.42, -64.5) mm, rotated rx -180 ry 0 rz 0.01 deg; joints [40.761, -43.969, 105.249, -135.702, 69.244, 161.77]
  MoveL 6953 to (-82.56, 264.15, -64.5) mm, rotated rx 180 ry 0 rz 0.01 deg; joints [40.458, -44.299, 105.999, -136.118, 69.445, 162.194]
  MoveC 6954 to (-83.27, 260.54, -64.5) mm, rotated rx -180 ry 0 rz 0.01 deg; joints [40.333, -44.37, 106.163, -136.268, 69.471, 162.308] to (-85.87, 257.93, -64.5) mm, rotated rx 180 ry 0 rz 0.01 deg; joints [40.19, -44.356, 106.136, -136.408, 69.415, 162.35]
  MoveC 6955 to (-88.46, 255.33, -64.5) mm, rotated rx -180 ry 0 rz 0.01 deg; joints [40.048, -44.341, 106.108, -136.549, 69.359, 162.393] to (-89.17, 251.72, -64.5) mm, rotated rx -180 ry 0 rz 0.01 deg; joints [39.923, -44.412, 106.27, -136.699, 69.385, 162.506]
  MoveL 6956 to (-82.15, 181.51, -64.5) mm, rotated rx 180 ry 0 rz 0.01 deg; joints [37.935, -46.344, 110.711, -139.326, 70.649, 165.002]
  MoveC 6957 to (-80.49, 176.35, -64.5) mm, rotated rx 180 ry 0 rz 0.01 deg; joints [37.811, -46.514, 111.105, -139.502, 70.784, 165.199] to (-76.85, 172.33, -64.5) mm, rotated rx -180 ry 0 rz 0.01 deg; joints [37.773, -46.719, 111.573, -139.601, 70.974, 165.394]
  MoveL 6958 to (-45.19, 149.58, -64.5) mm, rotated rx 180 ry 0 rz 0.01 deg; joints [37.832, -48.185, 114.948, -139.948, 72.447, 166.672]
  MoveC 6959 to (-43.06, 149.42, -64.5) mm, rotated rx 180 ry 0 rz 0.01 deg; joints [37.881, -48.251, 115.1, -139.916, 72.525, 166.715] to (-41.94, 151.24, -64.5) mm, rotated rx -180 ry 0 rz 0.01 deg; joints [37.97, -48.244, 115.08, -139.823, 72.538, 166.678]
  MoveL 6960 to (-41.95, 283.14, -64.5) mm, rotated rx 180 ry 0 rz 0.01 deg; joints [42.063, -45.051, 107.638, -134.731, 70.603, 162.287]
  MoveC 6961 to (-43.08, 285.86, -64.5) mm, rotated rx 180 ry 0 rz 0.01 deg; joints [42.112, -44.945, 107.397, -134.647, 70.525, 162.169] to (-45.8, 286.99, -64.5) mm, rotated rx 180 ry 0 rz 0.01 deg; joints [42.073, -44.833, 107.146, -134.651, 70.414, 162.077]
  MoveL 6962 to (-88.91, 286.99, -64.5) mm, rotated rx 180 ry 0 rz 0.01 deg; joints [40.966, -43.496, 104.185, -135.337, 68.893, 161.251]
  MoveC 6963 to (-91.45, 285.87, -64.5) mm, rotated rx 180 ry 0 rz 0.01 deg; joints [40.87, -43.445, 104.076, -135.418, 68.817, 161.243] to (-92.32, 283.23, -64.5) mm, rotated rx -180 ry 0 rz 0.01 deg; joints [40.771, -43.488, 104.174, -135.532, 68.824, 161.322]
  MoveL 6964 to (-89.17, 251.72, -64.5) mm, rotated rx 180 ry 0 rz 0.01 deg; joints [39.923, -44.412, 106.27, -136.699, 69.385, 162.506]
  MoveC 6965 to (-89.88, 248.11, -64.5) mm, rotated rx -180 ry 0 rz 0.01 deg; joints [39.797, -44.481, 106.43, -136.85, 69.411, 162.618] to (-92.47, 245.5, -64.5) mm, rotated rx -180 ry 0 rz 0.01 deg; joints [39.654, -44.466, 106.4, -136.99, 69.355, 162.66]
  MoveC 6966 to (-95.06, 242.89, -64.5) mm, rotated rx 180 ry 0 rz 0.01 deg; joints [39.511, -44.45, 106.369, -137.131, 69.298, 162.702] to (-95.78, 239.29, -64.5) mm, rotated rx 180 ry 0 rz 0.01 deg; joints [39.385, -44.518, 106.528, -137.282, 69.324, 162.814]
  MoveL 6967 to (-89.57, 177.23, -64.5) mm, rotated rx 180 ry 0 rz 0.01 deg; joints [37.616, -46.213, 110.424, -139.615, 70.44, 165.007]
  MoveC 6968 to (-87.91, 172.07, -64.5) mm, rotated rx -180 ry 0 rz 0.01 deg; joints [37.492, -46.383, 110.817, -139.792, 70.576, 165.203] to (-84.27, 168.05, -64.5) mm, rotated rx 180 ry 0 rz 0.01 deg; joints [37.452, -46.588, 111.286, -139.892, 70.767, 165.397]
  MoveL 6969 to (-37.38, 134.35, -64.5) mm, rotated rx -180 ry 0 rz 0.01 deg; joints [37.526, -48.747, 116.267, -140.409, 72.953, 167.276]
  MoveC 6970 to (-35.25, 134.19, -64.5) mm, rotated rx 180 ry 0 rz 0.01 deg; joints [37.576, -48.812, 116.419, -140.376, 73.031, 167.318] to (-34.13, 136.01, -64.5) mm, rotated rx 180 ry 0 rz 0.01 deg; joints [37.666, -48.806, 116.4, -140.282, 73.043, 167.282]
  MoveL 6971 to (-34.14, 290.95, -64.5) mm, rotated rx -180 ry 0 rz 0.01 deg; joints [42.497, -45.078, 107.686, -134.302, 70.76, 162.155]
  MoveC 6972 to (-35.27, 293.67, -64.5) mm, rotated rx 180 ry 0 rz 0.01 deg; joints [42.545, -44.972, 107.445, -134.219, 70.682, 162.036] to (-37.99, 294.8, -64.5) mm, rotated rx -180 ry 0 rz 0.01 deg; joints [42.506, -44.86, 107.194, -134.224, 70.572, 161.944]
  MoveL 6973 to (-97.54, 294.8, -64.5) mm, rotated rx 180 ry 0 rz 0.01 deg; joints [40.975, -43.009, 103.101, -135.164, 68.472, 160.796]
  MoveC 6974 to (-100.08, 293.67, -64.5) mm, rotated rx 180 ry 0 rz 0.01 deg; joints [40.879, -42.958, 102.991, -135.244, 68.396, 160.788] to (-100.95, 291.04, -64.5) mm, rotated rx 180 ry 0 rz 0.01 deg; joints [40.782, -43.001, 103.09, -135.358, 68.402, 160.868]
  MoveL 6975 to (-95.78, 239.29, -64.5) mm, rotated rx 180 ry 0 rz 0.01 deg; joints [39.385, -44.518, 106.528, -137.282, 69.324, 162.814]
  MoveC 6976 to (-96.49, 235.68, -64.5) mm, rotated rx 180 ry 0 rz 0.01 deg; joints [39.259, -44.587, 106.686, -137.433, 69.349, 162.925] to (-99.08, 233.07, -64.5) mm, rotated rx 180 ry 0 rz 0.01 deg; joints [39.116, -44.57, 106.653, -137.574, 69.292, 162.966]
  MoveC 6977 to (-101.67, 230.46, -64.5) mm, rotated rx -180 ry 0 rz 0.01 deg; joints [38.973, -44.552, 106.619, -137.714, 69.235, 163.007] to (-102.38, 226.85, -64.5) mm, rotated rx 180 ry 0 rz 0.01 deg; joints [38.846, -44.619, 106.774, -137.866, 69.26, 163.118]
  MoveL 6978 to (-96.99, 172.94, -64.5) mm, rotated rx 180 ry 0 rz 0.01 deg; joints [37.298, -46.079, 110.133, -139.902, 70.23, 165.011]
  MoveC 6979 to (-95.33, 167.78, -64.5) mm, rotated rx -180 ry 0 rz 0.01 deg; joints [37.173, -46.25, 110.525, -140.08, 70.366, 165.207] to (-91.69, 163.76, -64.5) mm, rotated rx 180 ry 0 rz 0.01 deg; joints [37.133, -46.455, 110.995, -140.182, 70.557, 165.401]
  MoveL 6980 to (-29.57, 119.11, -64.5) mm, rotated rx 180 ry 0 rz 0.01 deg; joints [37.214, -49.298, 117.572, -140.87, 73.46, 167.87]
  MoveC 6981 to (-27.44, 118.96, -64.5) mm, rotated rx 180 ry 0 rz 0.01 deg; joints [37.264, -49.363, 117.723, -140.836, 73.538, 167.911] to (-26.32, 120.78, -64.5) mm, rotated rx -180 ry 0 rz 0.01 deg; joints [37.354, -49.357, 117.704, -140.742, 73.55, 167.876]
  MoveL 6982 to (-26.33, 298.76, -64.5) mm, rotated rx -180 ry 0 rz 0.01 deg; joints [42.931, -45.102, 107.726, -133.872, 70.915, 162.02]
  MoveC 6983 to (-27.46, 301.48, -64.5) mm, rotated rx 180 ry 0 rz 0.01 deg; joints [42.979, -44.995, 107.484, -133.79, 70.837, 161.901] to (-30.18, 302.61, -64.5) mm, rotated rx 180 ry 0 rz 0.01 deg; joints [42.938, -44.884, 107.234, -133.796, 70.728, 161.809]
  MoveL 6984 to (-106.17, 302.61, -64.5) mm, rotated rx 180 ry 0 rz 0.01 deg; joints [40.984, -42.517, 102.007, -134.986, 68.049, 160.336]
  MoveC 6985 to (-108.71, 301.48, -64.5) mm, rotated rx 180 ry 0 rz 0.01 deg; joints [40.889, -42.465, 101.896, -135.064, 67.973, 160.327] to (-109.58, 298.85, -64.5) mm, rotated rx 180 ry 0 rz 0.01 deg; joints [40.792, -42.509, 101.997, -135.178, 67.978, 160.408]
  MoveL 6986 to (-102.38, 226.85, -64.5) mm, rotated rx -180 ry 0 rz 0.01 deg; joints [38.846, -44.619, 106.774, -137.866, 69.26, 163.118]
  MoveC 6987 to (-103.09, 223.27, -64.5) mm, rotated rx 180 ry 0 rz 0.01 deg; joints [38.72, -44.686, 106.927, -138.016, 69.285, 163.227] to (-105.66, 220.68, -64.5) mm, rotated rx 180 ry 0 rz 0.01 deg; joints [38.578, -44.667, 106.891, -138.156, 69.228, 163.267]
  MoveC 6988 to (-108.24, 218.1, -64.5) mm, rotated rx 180 ry 0 rz 0.01 deg; joints [38.436, -44.649, 106.854, -138.296, 69.17, 163.306] to (-108.95, 214.52, -64.5) mm, rotated rx -180 ry 0 rz 0.01 deg; joints [38.309, -44.714, 107.005, -138.447, 69.195, 163.415]
  MoveL 6989 to (-104.33, 167.77, -64.5) mm, rotated rx 180 ry 0 rz 0.01 deg; joints [36.955, -45.967, 109.89, -140.221, 70.034, 165.044]
  MoveC 6990 to (-102.92, 163.4, -64.5) mm, rotated rx 180 ry 0 rz 0.01 deg; joints [36.849, -46.111, 110.222, -140.373, 70.149, 165.21] to (-99.84, 160, -64.5) mm, rotated rx -180 ry 0 rz 0.01 deg; joints [36.814, -46.285, 110.62, -140.461, 70.312, 165.374]
  MoveL 6991 to (-21.76, 103.88, -64.5) mm, rotated rx 180 ry 0 rz 0.01 deg; joints [36.894, -49.84, 118.862, -141.332, 73.97, 168.454]
  MoveC 6992 to (-19.63, 103.73, -64.5) mm, rotated rx -180 ry 0 rz 0.01 deg; joints [36.944, -49.905, 119.012, -141.297, 74.048, 168.495] to (-18.51, 105.55, -64.5) mm, rotated rx -180 ry 0 rz 0.01 deg; joints [37.036, -49.899, 118.995, -141.201, 74.059, 168.461]
  MoveL 6993 to (-18.52, 306.57, -64.5) mm, rotated rx -180 ry 0 rz 0.01 deg; joints [43.365, -45.123, 107.759, -133.442, 71.068, 161.884]
  MoveC 6994 to (-19.65, 309.29, -64.5) mm, rotated rx 180 ry 0 rz 0.01 deg; joints [43.413, -45.016, 107.516, -133.361, 70.991, 161.764] to (-22.37, 310.42, -64.5) mm, rotated rx 180 ry 0 rz 0.01 deg; joints [43.371, -44.904, 107.267, -133.367, 70.882, 161.672]
  MoveL 6995 to (-115.32, 310.42, -64.5) mm, rotated rx 180 ry 0 rz 0.01 deg; joints [40.98, -42.001, 100.866, -134.809, 67.606, 159.859]
  MoveC 6996 to (-117.68, 309.34, -64.5) mm, rotated rx 180 ry 0 rz 0.01 deg; joints [40.892, -41.953, 100.764, -134.882, 67.535, 159.852] to (-118.39, 306.84, -64.5) mm, rotated rx -180 ry 0 rz 0.01 deg; joints [40.804, -41.999, 100.868, -134.988, 67.544, 159.931]
  MoveC 6997 to (-118.2, 305.7, -64.5) mm, rotated rx 180 ry 0 rz 0.01 deg; joints [40.776, -42.037, 100.952, -135.029, 67.567, 159.978] to (-117.98, 304.57, -64.5) mm, rotated rx 180 ry 0 rz 0.01 deg; joints [40.749, -42.076, 101.039, -135.07, 67.591, 160.025]
  MoveC 6998 to (-117.77, 303.43, -64.5) mm, rotated rx 180 ry 0 rz 0.01 deg; joints [40.722, -42.114, 101.125, -135.112, 67.614, 160.072] to (-117.62, 302.28, -64.5) mm, rotated rx 180 ry 0 rz 0.01 deg; joints [40.693, -42.151, 101.206, -135.154, 67.636, 160.118]
  MoveL 6999 to (-108.95, 214.52, -64.5) mm, rotated rx -180 ry 0 rz 0.01 deg; joints [38.309, -44.714, 107.005, -138.447, 69.195, 163.415]
  MoveC 7000 to (-109.65, 210.98, -64.5) mm, rotated rx -180 ry 0 rz 0.01 deg; joints [38.183, -44.777, 107.153, -138.596, 69.22, 163.521] to (-112.19, 208.43, -64.5) mm, rotated rx 180 ry 0 rz 0.01 deg; joints [38.043, -44.758, 107.114, -138.734, 69.162, 163.56]
  MoveC 7001 to (-114.74, 205.88, -64.5) mm, rotated rx 180 ry 0 rz 0.01 deg; joints [37.903, -44.738, 107.074, -138.872, 69.104, 163.598] to (-115.44, 202.34, -64.5) mm, rotated rx -180 ry 0 rz 0.01 deg; joints [37.776, -44.801, 107.22, -139.021, 69.129, 163.704]
  MoveL 7002 to (-111.86, 165.83, -64.5) mm, rotated rx -180 ry 0 rz 0.01 deg; joints [36.713, -45.772, 109.457, -140.414, 69.782, 164.97]
  MoveC 7003 to (-111.8, 164.89, -64.5) mm, rotated rx -180 ry 0 rz 0.01 deg; joints [36.684, -45.796, 109.512, -140.45, 69.798, 165.002] to (-111.81, 163.95, -64.5) mm, rotated rx -180 ry 0 rz 0.01 deg; joints [36.654, -45.817, 109.561, -140.488, 69.811, 165.032]
  MoveC 7004 to (-111.85, 163, -64.5) mm, rotated rx 180 ry 0 rz 0.01 deg; joints [36.623, -45.837, 109.608, -140.526, 69.823, 165.061] to (-111.89, 162.06, -64.5) mm, rotated rx 180 ry 0 rz 0.01 deg; joints [36.591, -45.857, 109.655, -140.564, 69.835, 165.091]
  MoveC 7005 to (-111.08, 158.66, -64.5) mm, rotated rx 180 ry 0 rz 0.01 deg; joints [36.501, -45.96, 109.893, -140.688, 69.914, 165.214] to (-108.53, 156.26, -64.5) mm, rotated rx -180 ry 0 rz 0.01 deg; joints [36.485, -46.096, 110.201, -140.744, 70.043, 165.337]
  MoveC 7006 to (-107.67, 155.82, -64.5) mm, rotated rx -180 ry 0 rz 0.01 deg; joints [36.491, -46.133, 110.285, -140.749, 70.082, 165.366] to (-106.81, 155.37, -64.5) mm, rotated rx 180 ry 0 rz 0.01 deg; joints [36.497, -46.17, 110.37, -140.753, 70.12, 165.396]
  MoveC 7007 to (-105.97, 154.9, -64.5) mm, rotated rx 180 ry 0 rz 0.01 deg; joints [36.502, -46.207, 110.454, -140.759, 70.158, 165.426] to (-105.17, 154.36, -64.5) mm, rotated rx 180 ry 0 rz 0.01 deg; joints [36.504, -46.245, 110.54, -140.768, 70.195, 165.458]
  MoveL 7008 to (-13.95, 88.65, -64.5) mm, rotated rx -180 ry 0 rz 0.01 deg; joints [36.567, -50.372, 120.138, -141.794, 74.481, 169.028]
  MoveC 7009 to (-11.82, 88.49, -64.5) mm, rotated rx -180 ry 0 rz 0.01 deg; joints [36.617, -50.436, 120.288, -141.758, 74.559, 169.069] to (-10.7, 90.32, -64.5) mm, rotated rx 180 ry 0 rz 0.01 deg; joints [36.71, -50.431, 120.272, -141.662, 74.57, 169.036]
  MoveL 7010 to (-10.71, 314.38, -64.5) mm, rotated rx 180 ry 0 rz 0.01 deg; joints [43.8, -45.14, 107.785, -133.011, 71.22, 161.746]
  MoveC 7011 to (-11.84, 317.1, -64.5) mm, rotated rx -180 ry 0 rz 0.01 deg; joints [43.846, -45.032, 107.541, -132.931, 71.142, 161.625] to (-14.56, 318.23, -64.5) mm, rotated rx 180 ry 0 rz 0.01 deg; joints [43.804, -44.921, 107.293, -132.938, 71.034, 161.533]
  MoveL 7012 to (-125.79, 318.23, -64.5) mm, rotated rx 180 ry 0 rz 0.01 deg; joints [40.944, -41.434, 99.617, -134.643, 67.112, 159.347]
  MoveC 7013 to (-127.94, 317.15, -64.5) mm, rotated rx 180 ry 0 rz 0.01 deg; joints [40.861, -41.393, 99.528, -134.712, 67.048, 159.344] to (-128.36, 314.78, -64.5) mm, rotated rx -180 ry 0 rz 0.01 deg; joints [40.785, -41.446, 99.647, -134.809, 67.066, 159.426]
  MoveC 7014 to (-127.46, 311.75, -64.5) mm, rotated rx 180 ry 0 rz 0.01 deg; joints [40.721, -41.561, 99.903, -134.915, 67.141, 159.56] to (-126.58, 308.72, -64.5) mm, rotated rx -180 ry 0 rz 0.01 deg; joints [40.657, -41.675, 100.157, -135.022, 67.216, 159.693]
  MoveC 7015 to (-125.82, 305.65, -64.5) mm, rotated rx 180 ry 0 rz 0.01 deg; joints [40.589, -41.786, 100.404, -135.131, 67.287, 159.825] to (-125.27, 302.53, -64.5) mm, rotated rx 180 ry 0 rz 0.01 deg; joints [40.513, -41.89, 100.637, -135.244, 67.351, 159.953]
  MoveL 7016 to (-115.44, 202.34, -64.5) mm, rotated rx 180 ry 0 rz 0.01 deg; joints [37.776, -44.801, 107.22, -139.021, 69.129, 163.704]
  MoveC 7017 to (-116.14, 198.81, -64.5) mm, rotated rx 180 ry 0 rz 0.01 deg; joints [37.65, -44.863, 107.365, -139.17, 69.153, 163.809] to (-118.68, 196.27, -64.5) mm, rotated rx -180 ry 0 rz 0.01 deg; joints [37.51, -44.842, 107.323, -139.308, 69.095, 163.847]
  MoveC 7018 to (-121.22, 193.73, -64.5) mm, rotated rx -180 ry 0 rz 0.01 deg; joints [37.37, -44.821, 107.28, -139.445, 69.036, 163.884] to (-121.92, 190.2, -64.5) mm, rotated rx -180 ry 0 rz 0.01 deg; joints [37.244, -44.882, 107.423, -139.595, 69.06, 163.988]
  MoveL 7019 to (-119.46, 165.07, -64.5) mm, rotated rx 180 ry 0 rz 0.01 deg; joints [36.508, -45.547, 108.953, -140.557, 69.51, 164.856]
  MoveC 7020 to (-119.39, 162.68, -64.5) mm, rotated rx 180 ry 0 rz 0.01 deg; joints [36.434, -45.603, 109.085, -140.651, 69.546, 164.935] to (-119.65, 160.31, -64.5) mm, rotated rx 180 ry 0 rz 0.01 deg; joints [36.351, -45.649, 109.192, -140.75, 69.57, 165.006]
  MoveC 7021 to (-120.17, 157.98, -64.5) mm, rotated rx 180 ry 0 rz 0.01 deg; joints [36.264, -45.685, 109.277, -140.851, 69.584, 165.071] to (-120.88, 155.7, -64.5) mm, rotated rx 180 ry 0 rz 0.01 deg; joints [36.174, -45.714, 109.346, -140.952, 69.59, 165.131]
  MoveC 7022 to (-120.68, 153.21, -64.5) mm, rotated rx 180 ry 0 rz 0.01 deg; joints [36.099, -45.777, 109.491, -141.049, 69.633, 165.215] to (-118.68, 151.7, -64.5) mm, rotated rx -180 ry 0 rz 0.01 deg; joints [36.097, -45.875, 109.714, -141.08, 69.729, 165.299]
  MoveC 7023 to (-117.05, 151.3, -64.5) mm, rotated rx 180 ry 0 rz 0.01 deg; joints [36.122, -45.936, 109.852, -141.071, 69.796, 165.341] to (-115.44, 150.84, -64.5) mm, rotated rx 180 ry 0 rz 0.01 deg; joints [36.146, -45.997, 109.991, -141.065, 69.863, 165.384]
  MoveC 7024 to (-113.85, 150.3, -64.5) mm, rotated rx 180 ry 0 rz 0.01 deg; joints [36.166, -46.06, 110.133, -141.063, 69.93, 165.43] to (-112.31, 149.64, -64.5) mm, rotated rx 180 ry 0 rz 0.01 deg; joints [36.181, -46.124, 110.278, -141.066, 69.997, 165.479]
  MoveC 7025 to (-111.61, 149.31, -64.5) mm, rotated rx -180 ry 0 rz 0.01 deg; joints [36.187, -46.154, 110.345, -141.069, 70.028, 165.502] to (-110.93, 148.97, -64.5) mm, rotated rx 180 ry 0 rz 0.01 deg; joints [36.192, -46.183, 110.411, -141.072, 70.058, 165.525]
  MoveC 7026 to (-110.26, 148.59, -64.5) mm, rotated rx 180 ry 0 rz 0.01 deg; joints [36.196, -46.213, 110.479, -141.077, 70.089, 165.549] to (-109.62, 148.17, -64.5) mm, rotated rx -180 ry 0 rz 0.01 deg; joints [36.197, -46.242, 110.546, -141.084, 70.119, 165.574]
  MoveL 7027 to (-6.14, 73.42, -64.5) mm, rotated rx 180 ry 0 rz 0.01 deg; joints [36.232, -50.894, 121.401, -142.258, 74.995, 169.593]
  MoveC 7028 to (-4.01, 73.26, -64.5) mm, rotated rx -180 ry 0 rz 0.01 deg; joints [36.282, -50.957, 121.55, -142.221, 75.073, 169.634] to (-2.89, 75.09, -64.5) mm, rotated rx -180 ry 0 rz 0.01 deg; joints [36.376, -50.953, 121.535, -142.124, 75.084, 169.602]
  MoveL 7029 to (-2.9, 322.19, -64.5) mm, rotated rx 180 ry 0 rz 0.01 deg; joints [44.235, -45.153, 107.802, -132.58, 71.369, 161.606]
  MoveC 7030 to (-4.03, 324.91, -64.5) mm, rotated rx -180 ry 0 rz 0.01 deg; joints [44.281, -45.045, 107.558, -132.501, 71.292, 161.485] to (-6.75, 326.04, -64.5) mm, rotated rx 180 ry 0 rz 0.01 deg; joints [44.238, -44.935, 107.31, -132.509, 71.185, 161.392]
  MoveL 7031 to (-138.54, 326.04, -64.5) mm, rotated rx -180 ry 0 rz 0.01 deg; joints [40.854, -40.782, 98.186, -134.496, 66.531, 158.78]
  MoveC 7032 to (-140.47, 324.92, -64.5) mm, rotated rx -180 ry 0 rz 0.01 deg; joints [40.776, -40.748, 98.113, -134.563, 66.474, 158.783] to (-140.48, 322.69, -64.5) mm, rotated rx 180 ry 0 rz 0.01 deg; joints [40.714, -40.812, 98.255, -134.65, 66.505, 158.869]
  MoveC 7033 to (-138.6, 319.3, -64.5) mm, rotated rx -180 ry 0 rz 0.01 deg; joints [40.664, -40.973, 98.609, -134.759, 66.623, 159.04] to (-136.81, 315.86, -64.5) mm, rotated rx 180 ry 0 rz 0.01 deg; joints [40.611, -41.131, 98.959, -134.871, 66.737, 159.209]
  MoveC 7034 to (-135.28, 312.29, -64.5) mm, rotated rx -180 ry 0 rz 0.01 deg; joints [40.547, -41.283, 99.296, -134.991, 66.844, 159.377] to (-134.21, 308.56, -64.5) mm, rotated rx -180 ry 0 rz 0.01 deg; joints [40.468, -41.424, 99.608, -135.123, 66.936, 159.542]
  MoveC 7035 to (-133.78, 306.63, -64.5) mm, rotated rx 180 ry 0 rz 0.01 deg; joints [40.424, -41.492, 99.761, -135.193, 66.979, 159.624] to (-133.37, 304.69, -64.5) mm, rotated rx -180 ry 0 rz 0.01 deg; joints [40.379, -41.56, 99.912, -135.264, 67.021, 159.706]
  MoveC 7036 to (-133.02, 302.73, -64.5) mm, rotated rx 180 ry 0 rz 0.01 deg; joints [40.332, -41.626, 100.059, -135.335, 67.062, 159.787] to (-132.77, 300.77, -64.5) mm, rotated rx 180 ry 0 rz 0.01 deg; joints [40.282, -41.689, 100.199, -135.409, 67.098, 159.866]
  MoveL 7037 to (-121.92, 190.2, -64.5) mm, rotated rx 180 ry 0 rz 0.01 deg; joints [37.244, -44.882, 107.423, -139.595, 69.06, 163.988]
  MoveL 7038 to (-121.71, 189.61, -64.33) mm, rotated rx 180 ry 0 rz 0.01 deg; joints [37.23, -44.912, 107.472, -139.613, 69.071, 164.006]
  MoveL 7039 to (-121.38, 189.28, -63.87) mm, rotated rx 180 ry 0 rz 0.01 deg; joints [37.227, -44.956, 107.517, -139.616, 69.07, 164.008]
  MoveL 7040 to (-121.23, 189.19, -63.23) mm, rotated rx 180 ry 0 rz 0.01 deg; joints [37.228, -44.998, 107.536, -139.611, 69.054, 163.993]
  Set speed (1000.0 mm/s)
  MoveL 7041 to (-121.23, 189.19, 11) mm, rotated rx -180 ry 0 rz 0.01 deg; joints [37.191, -48.976, 107.829, -138.657, 66.254, 161.4]
  Set speed (1000.0 mm/s)
  MoveL 7042 to (-206.45, 109.97, 11) mm, rotated rx -180 ry 0 rz 0.01 deg; joints [32.751, -47.821, 105.6, -142.959, 63.949, 162.644]
  Set speed (1000.0 mm/s)
  MoveL 7043 to (-206.45, 109.97, -42.73) mm, rotated rx 180 ry 0 rz 0.01 deg; joints [32.781, -45.02, 105.432, -143.661, 66.069, 164.366]
  Set speed (100.0 mm/s)
  MoveL 7044 to (-206.47, 109.81, -43.35) mm, rotated rx -180 ry 0 rz 0.01 deg; joints [32.776, -44.99, 105.435, -143.675, 66.095, 164.39]
  MoveL 7045 to (-206.5, 109.37, -43.82) mm, rotated rx 180 ry 0 rz 0.01 deg; joints [32.761, -44.975, 105.453, -143.7, 66.117, 164.418]
  MoveL 7046 to (-206.48, 108.75, -44) mm, rotated rx 180 ry 0 rz 0.01 deg; joints [32.742, -44.979, 105.484, -143.727, 66.133, 164.444]
  MoveL 7047 to (-202.46, 103.51, -44.24) mm, rotated rx 180 ry 0 rz 0.01 deg; joints [32.655, -45.224, 106.052, -143.901, 66.369, 164.69]
  MoveL 7048 to (-196.05, 105.1, -44.49) mm, rotated rx -180 ry 0 rz 0.01 deg; joints [32.842, -45.403, 106.465, -143.766, 66.611, 164.76]
  MoveL 7049 to (-194.93, 111.61, -44.73) mm, rotated rx 180 ry 0 rz 0.01 deg; joints [33.079, -45.286, 106.226, -143.488, 66.581, 164.581]
  MoveL 7050 to (-200.45, 115.24, -44.98) mm, rotated rx -180 ry 0 rz 0.01 deg; joints [33.08, -44.998, 105.62, -143.404, 66.326, 164.374]
  MoveL 7051 to (-205.99, 111.64, -45.22) mm, rotated rx 180 ry 0 rz 0.01 deg; joints [32.847, -44.868, 105.372, -143.617, 66.162, 164.398]
  MoveL 7052 to (-204.9, 105.12, -45.46) mm, rotated rx 180 ry 0 rz 0.01 deg; joints [32.657, -45.037, 105.777, -143.877, 66.298, 164.632]
  MoveL 7053 to (-198.5, 103.5, -45.71) mm, rotated rx -180 ry 0 rz 0.01 deg; joints [32.739, -45.286, 106.349, -143.874, 66.582, 164.805]
  MoveL 7054 to (-194.45, 108.72, -45.95) mm, rotated rx -180 ry 0 rz 0.01 deg; joints [32.995, -45.301, 106.4, -143.616, 66.684, 164.719]
  MoveL 7055 to (-197.61, 114.52, -46.2) mm, rotated rx -180 ry 0 rz 0.01 deg; joints [33.117, -45.049, 105.868, -143.416, 66.494, 164.486]
  MoveL 7056 to (-204.19, 113.95, -46.44) mm, rotated rx -180 ry 0 rz 0.01 deg; joints [32.96, -44.816, 105.388, -143.516, 66.251, 164.393]
  MoveL 7057 to (-206.31, 107.7, -46.68) mm, rotated rx -180 ry 0 rz 0.01 deg; joints [32.713, -44.865, 105.535, -143.8, 66.257, 164.563]
  MoveL 7058 to (-201.42, 103.25, -46.93) mm, rotated rx 180 ry 0 rz 0.01 deg; joints [32.67, -45.123, 106.13, -143.932, 66.518, 164.798]
  MoveL 7059 to (-195.39, 105.94, -47.17) mm, rotated rx -180 ry 0 rz 0.01 deg; joints [32.885, -45.263, 106.458, -143.755, 66.731, 164.828]
  MoveL 7060 to (-195.44, 112.55, -47.42) mm, rotated rx 180 ry 0 rz 0.01 deg; joints [33.1, -45.104, 106.125, -143.487, 66.653, 164.625]
  MoveL 7061 to (-201.51, 115.15, -47.66) mm, rotated rx 180 ry 0 rz 0.01 deg; joints [33.056, -44.819, 105.528, -143.452, 66.388, 164.44]
  MoveL 7062 to (-206.33, 110.63, -47.9) mm, rotated rx -180 ry 0 rz 0.01 deg; joints [32.808, -44.735, 105.38, -143.694, 66.265, 164.506]
  MoveL 7063 to (-204.12, 104.41, -48.15) mm, rotated rx 180 ry 0 rz 0.01 deg; joints [32.652, -44.937, 105.858, -143.929, 66.443, 164.751]
  MoveL 7064 to (-197.53, 103.94, -48.39) mm, rotated rx 180 ry 0 rz 0.01 deg; joints [32.775, -45.166, 106.387, -143.877, 66.72, 164.891]
  MoveL 7065 to (-194.46, 109.79, -48.64) mm, rotated rx -180 ry 0 rz 0.01 deg; joints [33.031, -45.133, 106.331, -143.603, 66.774, 164.768]
  MoveL 7066 to (-198.59, 114.94, -48.88) mm, rotated rx -180 ry 0 rz 0.01 deg; joints [33.112, -44.862, 105.756, -143.442, 66.554, 164.537]
  MoveL 7067 to (-204.97, 113.22, -49.13) mm, rotated rx -180 ry 0 rz 0.01 deg; joints [32.922, -44.661, 105.349, -143.587, 66.333, 164.485]
  MoveL 7068 to (-205.95, 106.69, -49.37) mm, rotated rx 180 ry 0 rz 0.01 deg; joints [32.689, -44.757, 105.597, -143.869, 66.388, 164.683]
  MoveL 7069 to (-200.36, 103.18, -49.61) mm, rotated rx 180 ry 0 rz 0.01 deg; joints [32.691, -45.018, 106.2, -143.954, 66.665, 164.902]
  MoveL 7070 to (-194.9, 106.89, -49.86) mm, rotated rx 180 ry 0 rz 0.01 deg; joints [32.928, -45.116, 106.434, -143.742, 66.842, 164.889]
  MoveL 7071 to (-196.11, 113.38, -50.1) mm, rotated rx -180 ry 0 rz 0.01 deg; joints [33.114, -44.918, 106.017, -143.492, 66.719, 164.669]
  MoveL 7072 to (-202.54, 114.87, -50.35) mm, rotated rx 180 ry 0 rz 0.01 deg; joints [33.027, -44.646, 105.447, -143.506, 66.454, 164.513]
  MoveL 7073 to (-206.49, 109.57, -50.59) mm, rotated rx 180 ry 0 rz 0.01 deg; joints [32.772, -44.61, 105.405, -143.771, 66.376, 164.618]
  MoveL 7074 to (-203.21, 103.84, -50.83) mm, rotated rx -180 ry 0 rz 0.01 deg; joints [32.654, -44.837, 105.94, -143.973, 66.59, 164.867]
  MoveL 7075 to (-196.65, 104.54, -51.08) mm, rotated rx 180 ry 0 rz 0.01 deg; joints [32.815, -45.04, 106.409, -143.873, 66.851, 164.969]
  MoveL 7076 to (-194.66, 110.84, -51.32) mm, rotated rx 180 ry 0 rz 0.01 deg; joints [33.063, -44.959, 106.248, -143.594, 66.857, 164.813]
  MoveL 7077 to (-199.63, 115.18, -51.57) mm, rotated rx 180 ry 0 rz 0.01 deg; joints [33.099, -44.676, 105.648, -143.475, 66.612, 164.593]
  MoveL 7078 to (-205.6, 112.37, -51.81) mm, rotated rx -180 ry 0 rz 0.01 deg; joints [32.882, -44.514, 105.327, -143.66, 66.421, 164.582]
  MoveL 7079 to (-205.42, 105.77, -52.05) mm, rotated rx 180 ry 0 rz 0.01 deg; joints [32.671, -44.652, 105.667, -143.933, 66.524, 164.803]
  MoveL 7080 to (-199.3, 103.29, -52.3) mm, rotated rx -180 ry 0 rz 0.01 deg; joints [32.719, -44.908, 106.26, -143.968, 66.81, 164.998]
  MoveL 7081 to (-194.57, 107.91, -52.54) mm, rotated rx 180 ry 0 rz 0.01 deg; joints [32.97, -44.96, 106.392, -143.727, 66.946, 164.945]
  MoveL 7082 to (-196.91, 114.08, -52.79) mm, rotated rx -180 ry 0 rz 0.01 deg; joints [33.121, -44.73, 105.904, -143.503, 66.781, 164.714]
  MoveL 7083 to (-203.51, 114.42, -53.03) mm, rotated rx 180 ry 0 rz 0.01 deg; joints [32.993, -44.478, 105.379, -143.567, 66.524, 164.592]
  MoveL 7084 to (-206.46, 108.51, -53.27) mm, rotated rx 180 ry 0 rz 0.01 deg; joints [32.739, -44.49, 105.444, -143.846, 66.494, 164.734]
  MoveL 7085 to (-202.22, 103.44, -53.52) mm, rotated rx 180 ry 0 rz 0.01 deg; joints [32.663, -44.737, 106.02, -144.01, 66.739, 164.978]
  MoveL 7086 to (-195.88, 105.28, -53.76) mm, rotated rx 180 ry 0 rz 0.01 deg; joints [32.857, -44.906, 106.414, -143.864, 66.976, 165.041]
  MoveL 7087 to (-195.03, 111.83, -54.01) mm, rotated rx 180 ry 0 rz 0.01 deg; joints [33.089, -44.78, 106.153, -143.588, 66.932, 164.857]
  MoveL 7088 to (-200.69, 115.24, -54.25) mm, rotated rx 180 ry 0 rz 0.01 deg; joints [33.08, -44.494, 105.547, -143.516, 66.672, 164.654]
  MoveL 7089 to (-206.08, 111.41, -54.49) mm, rotated rx 180 ry 0 rz 0.01 deg; joints [32.842, -44.375, 105.321, -143.736, 66.518, 164.685]
  MoveL 7090 to (-204.74, 104.95, -54.74) mm, rotated rx -180 ry 0 rz 0.01 deg; joints [32.66, -44.55, 105.744, -143.99, 66.666, 164.922]
  MoveL 7091 to (-198.27, 103.59, -54.98) mm, rotated rx 180 ry 0 rz 0.01 deg; joints [32.752, -44.793, 106.307, -143.975, 66.951, 165.089]
  MoveL 7092 to (-194.44, 108.96, -55.23) mm, rotated rx 180 ry 0 rz 0.01 deg; joints [33.009, -44.797, 106.334, -143.713, 67.041, 164.996]
  MoveL 7093 to (-197.83, 114.63, -55.47) mm, rotated rx 180 ry 0 rz 0.01 deg; joints [33.121, -44.542, 105.79, -143.522, 66.841, 164.762]
  MoveL 7094 to (-204.38, 113.8, -55.71) mm, rotated rx 180 ry 0 rz 0.01 deg; joints [32.956, -44.318, 105.326, -143.633, 66.6, 164.677]
  MoveL 7095 to (-206.24, 107.46, -55.96) mm, rotated rx 180 ry 0 rz 0.01 deg; joints [32.711, -44.377, 105.496, -143.917, 66.619, 164.852]
  MoveL 7096 to (-201.18, 103.22, -56.2) mm, rotated rx 180 ry 0 rz 0.01 deg; joints [32.679, -44.633, 106.094, -144.037, 66.887, 165.085]
  MoveL 7097 to (-195.26, 106.15, -56.45) mm, rotated rx -180 ry 0 rz 0.01 deg; joints [32.9, -44.763, 106.402, -143.852, 67.093, 165.106]
  MoveL 7098 to (-195.58, 112.75, -56.69) mm, rotated rx 180 ry 0 rz 0.01 deg; joints [33.108, -44.596, 106.048, -143.588, 67.002, 164.9]
  MoveL 7099 to (-201.75, 115.1, -56.93) mm, rotated rx 180 ry 0 rz 0.01 deg; joints [33.054, -44.316, 105.455, -143.564, 66.734, 164.72]
  MoveL 7100 to (-206.38, 110.39, -57.18) mm, rotated rx 180 ry 0 rz 0.01 deg; joints [32.804, -44.243, 105.332, -143.812, 66.622, 164.793]
  MoveL 7101 to (-203.92, 104.26, -57.42) mm, rotated rx -180 ry 0 rz 0.01 deg; joints [32.656, -44.449, 105.824, -144.039, 66.811, 165.039]
  MoveL 7102 to (-197.32, 104.06, -57.67) mm, rotated rx -180 ry 0 rz 0.01 deg; joints [32.789, -44.671, 106.34, -143.975, 67.086, 165.172]
  MoveL 7103 to (-194.49, 110.03, -57.91) mm, rotated rx -180 ry 0 rz 0.01 deg; joints [33.044, -44.627, 106.26, -143.7, 67.128, 165.042]
  MoveL 7104 to (-198.82, 115.01, -58.15) mm, rotated rx 180 ry 0 rz 0.01 deg; joints [33.114, -44.355, 105.677, -143.549, 66.899, 164.813]
  MoveL 7105 to (-205.13, 113.04, -58.4) mm, rotated rx 180 ry 0 rz 0.01 deg; joints [32.917, -44.164, 105.289, -143.704, 66.683, 164.769]
  MoveL 7106 to (-205.84, 106.47, -58.64) mm, rotated rx 180 ry 0 rz 0.01 deg; joints [32.689, -44.268, 105.558, -143.984, 66.751, 164.971]
  MoveL 7107 to (-200.11, 103.19, -58.89) mm, rotated rx 180 ry 0 rz 0.01 deg; joints [32.702, -44.526, 106.16, -144.057, 67.034, 165.186]
  MoveL 7108 to (-194.81, 107.12, -59.13) mm, rotated rx -180 ry 0 rz 0.01 deg; joints [32.943, -44.613, 106.372, -143.837, 67.202, 165.165]
